LIN {X 0,Y 231.283,Z 816.098,A -85,B 0,C 180,E1 32036.153,E2 32036.153} C_VEL
LIN {X 0,Y 232.3,Z 814.541,A -85,B 0,C 180,E1 32036.256,E2 32036.256} C_VEL
LIN {X 0,Y 232.997,Z 811.859,A -85,B 0,C 180,E1 32038.132,E2 32038.132} C_VEL
LIN {X 0,Y 233.164,Z 810.301,A -85,B 0,C 180,E1 32039.995,E2 32039.995} C_VEL
LIN {X 0,Y 231.964,Z 810.617,A -85,B 0,C 180,E1 32043.74,E2 32043.74} C_VEL
LIN {X 0,Y 228.908,Z 815.493,A -85,B 0,C 180,E1 32049.516,E2 32049.516} C_VEL
LIN {X 0,Y 226.036,Z 820.81,A -85,B 0,C 180,E1 32052.805,E2 32052.805} C_VEL
LIN {X 0,Y 201.465,Z 849.972,A -85,B 0,C 180,E1 32056.439,E2 32056.439} C_VEL
LIN {X 0,Y 175.055,Z 874.28,A -85,B 0,C 180,E1 32061.454,E2 32061.454} C_VEL
LIN {X 0,Y 147.098,Z 894.32,A -85,B 0,C 180,E1 32068.856,E2 32068.856} C_VEL
LIN {X 0,Y 119.761,Z 909.714,A -85,B 0,C 180,E1 32080.583,E2 32080.583} C_VEL
LIN {X 0,Y 99.708,Z 918.948,A -85,B 0,C 180,E1 32096.749,E2 32096.749} C_VEL
LIN {X 0,Y 88.361,Z 923.461,A -85,B 0,C 180,E1 32120.099,E2 32120.099} C_VEL
LIN {X 0,Y 88.441,Z 923.431,A -85,B 0,C 180,E1 32139.837,E2 32139.837} C_VEL
LIN {X 0,Y 99.926,Z 918.782,A -85,B 0,C 180,E1 32163.44,E2 32163.44} C_VEL
LIN {X 0,Y 119.785,Z 909.607,A -85,B 0,C 180,E1 32179.342,E2 32179.342} C_VEL
LIN {X 0,Y 119.619,Z 909.301,A -85,B 0,C 180,E1 32180.724,E2 32180.724} C_VEL
LIN {X 0,Y 90.219,Z 920.421,A -85,B 0,C 180,E1 32221.835,E2 32221.835} C_VEL
LIN {X 0,Y 87.807,Z 924.074,A -85,B 0,C 180,E1 32232.793,E2 32232.793} C_VEL
LIN {X 0,Y 88.883,Z 927.566,A -85,B 0,C 180,E1 32243.903,E2 32243.903} C_VEL
LIN {X 0,Y 99.549,Z 930.781,A -85,B 0,C 180,E1 32256.148,E2 32256.148} C_VEL
LIN {X 0,Y 97.42,Z 932.429,A -85,B 0,C 180,E1 32258.992,E2 32258.992} C_VEL
LIN {X 0,Y 80.593,Z 941.329,A -85,B 0,C 180,E1 32281.998,E2 32281.998} C_VEL
LIN {X 0,Y 77.652,Z 944.052,A -85,B 0,C 180,E1 32298.779,E2 32298.779} C_VEL
LIN {X 0,Y 78.572,Z 944.794,A -85,B 0,C 180,E1 32310.03,E2 32310.03} C_VEL
LIN {X 0,Y 78.579,Z 942.435,A -85,B 0,C 180,E1 32332.717,E2 32332.717} C_VEL
LIN {X 0,Y 92.775,Z 933.853,A -85,B 0,C 180,E1 32359.206,E2 32359.206} C_VEL
LIN {X 0,Y 118.649,Z 919.574,A -85,B 0,C 180,E1 32376.148,E2 32376.148} C_VEL
LIN {X 0,Y 147.805,Z 900.768,A -85,B 0,C 180,E1 32385.844,E2 32385.844} C_VEL
LIN {X 0,Y 177.973,Z 876.597,A -85,B 0,C 180,E1 32391.869,E2 32391.869} C_VEL
LIN {X 0,Y 206.02,Z 847.904,A -85,B 0,C 180,E1 32395.688,E2 32395.688} C_VEL
LIN {X 0,Y 227.481,Z 820.1,A -85,B 0,C 180,E1 32397.863,E2 32397.863} C_VEL
LIN {X 0,Y 228.556,Z 817.821,A -85,B 0,C 180,E1 32398.934,E2 32398.934} C_VEL
LIN {X 0,Y 228.688,Z 816.963,A -85,B 0,C 180,E1 32399.995,E2 32399.995} C_VEL
LIN {X 0,Y 227.313,Z 817.302,A -85,B 0,C 180,E1 32403.816,E2 32403.816} C_VEL
LIN {X 0,Y 223.822,Z 822.315,A -85,B 0,C 180,E1 32409.605,E2 32409.605} C_VEL
LIN {X 0,Y 221.659,Z 825.693,A -85,B 0,C 180,E1 32411.2,E2 32411.2} C_VEL
LIN {X 0,Y 195.972,Z 854.587,A -85,B 0,C 180,E1 32414.832,E2 32414.832} C_VEL
LIN {X 0,Y 167.376,Z 879.131,A -85,B 0,C 180,E1 32420.037,E2 32420.037} C_VEL
LIN {X 0,Y 140.432,Z 897.198,A -85,B 0,C 180,E1 32427.072,E2 32427.072} C_VEL
LIN {X 0,Y 112.214,Z 911.987,A -85,B 0,C 180,E1 32439.033,E2 32439.033} C_VEL
LIN {X 0,Y 92.464,Z 920.215,A -85,B 0,C 180,E1 32454.982,E2 32454.982} C_VEL
LIN {X 0,Y 80.648,Z 924.449,A -85,B 0,C 180,E1 32479.141,E2 32479.141} C_VEL
LIN {X 0,Y 80.725,Z 924.423,A -85,B 0,C 180,E1 32500.788,E2 32500.788} C_VEL
LIN {X 0,Y 92.642,Z 920.094,A -85,B 0,C 180,E1 32525.175,E2 32525.175} C_VEL
LIN {X 0,Y 109.719,Z 912.985,A -85,B 0,C 180,E1 32539.39,E2 32539.39} C_VEL
LIN {X 0,Y 108.72,Z 912.974,A -85,B 0,C 180,E1 32541.182,E2 32541.182} C_VEL
LIN {X 0,Y 88.883,Z 927.566,A -85,B 0,C 180,E1 32603.903,E2 32603.903} C_VEL
LIN {X 0,Y 91.046,Z 929.778,A -85,B 0,C 180,E1 32610.655,E2 32610.655} C_VEL
LIN {X 0,Y 89.329,Z 932.69,A -85,B 0,C 180,E1 32617.152,E2 32617.152} C_VEL
LIN {X 0,Y 87.849,Z 933.503,A -85,B 0,C 180,E1 32618.803,E2 32618.803} C_VEL
LIN {X 0,Y 71.627,Z 941.461,A -85,B 0,C 180,E1 32645.008,E2 32645.008} C_VEL
LIN {X 0,Y 70.618,Z 943.791,A -85,B 0,C 180,E1 32670.034,E2 32670.034} C_VEL
LIN {X 0,Y 71.144,Z 941.405,A -85,B 0,C 180,E1 32695.248,E2 32695.248} C_VEL
LIN {X 0,Y 87.583,Z 932.779,A -85,B 0,C 180,E1 32723.316,E2 32723.316} C_VEL
LIN {X 0,Y 115.54,Z 918.483,A -85,B 0,C 180,E1 32739.919,E2 32739.919} C_VEL
LIN {X 0,Y 146.614,Z 899.19,A -85,B 0,C 180,E1 32749.136,E2 32749.136} C_VEL
LIN {X 0,Y 178.554,Z 874.062,A -85,B 0,C 180,E1 32754.74,E2 32754.74} C_VEL
LIN {X 0,Y 206.65,Z 845.496,A -85,B 0,C 180,E1 32758.072,E2 32758.072} C_VEL
LIN {X 0,Y 222.734,Z 825.385,A -85,B 0,C 180,E1 32759.528,E2 32759.528} C_VEL
LIN {X 0,Y 223.946,Z 823.43,A -85,B 0,C 180,E1 32759.995,E2 32759.995} C_VEL
LIN {X 0,Y 222.493,Z 823.879,A -85,B 0,C 180,E1 32763.899,E2 32763.899} C_VEL
LIN {X 0,Y 219.282,Z 827.949,A -85,B 0,C 180,E1 32768.768,E2 32768.768} C_VEL
LIN {X 0,Y 217.386,Z 830.343,A -85,B 0,C 180,E1 32769.537,E2 32769.537} C_VEL
LIN {X 0,Y 190.615,Z 858.942,A -85,B 0,C 180,E1 32773.101,E2 32773.101} C_VEL
LIN {X 0,Y 161.481,Z 882.675,A -85,B 0,C 180,E1 32778.139,E2 32778.139} C_VEL
LIN {X 0,Y 130.785,Z 901.732,A -85,B 0,C 180,E1 32786.079,E2 32786.079} C_VEL
LIN {X 0,Y 102.133,Z 915.175,A -85,B 0,C 180,E1 32798.806,E2 32798.806} C_VEL
LIN {X 0,Y 82.386,Z 922.477,A -85,B 0,C 180,E1 32816.478,E2 32816.478} C_VEL
LIN {X 0,Y 72.949,Z 925.439,A -85,B 0,C 180,E1 32837.979,E2 32837.979} C_VEL
LIN {X 0,Y 73.048,Z 925.413,A -85,B 0,C 180,E1 32861.938,E2 32861.938} C_VEL
LIN {X 0,Y 86.324,Z 921.102,A -85,B 0,C 180,E1 32888.188,E2 32888.188} C_VEL
LIN {X 0,Y 99.662,Z 916.141,A -85,B 0,C 180,E1 32899.442,E2 32899.442} C_VEL
LIN {X 0,Y 97.848,Z 916.351,A -85,B 0,C 180,E1 32901.751,E2 32901.751} C_VEL
LIN {X 0,Y 90.297,Z 932.103,A -85,B 0,C 180,E1 32975.972,E2 32975.972} C_VEL
LIN {X 0,Y 87.849,Z 933.503,A -85,B 0,C 180,E1 32978.803,E2 32978.803} C_VEL
LIN {X 0,Y 75.565,Z 937.247,A -85,B 0,C 180,E1 32987.238,E2 32987.238} C_VEL
LIN {X 0,Y 65.402,Z 939.87,A -85,B 0,C 180,E1 32998.741,E2 32998.741} C_VEL
LIN {X 0,Y 62.681,Z 942.791,A -85,B 0,C 180,E1 33030.038,E2 33030.038} C_VEL
LIN {X 0,Y 63.847,Z 940.368,A -85,B 0,C 180,E1 33058.378,E2 33058.378} C_VEL
LIN {X 0,Y 82.635,Z 931.823,A -85,B 0,C 180,E1 33087.678,E2 33087.678} C_VEL
LIN {X 0,Y 113.083,Z 917.306,A -85,B 0,C 180,E1 33103.951,E2 33103.951} C_VEL
LIN {X 0,Y 145.282,Z 898.069,A -85,B 0,C 180,E1 33112.343,E2 33112.343} C_VEL
LIN {X 0,Y 177.269,Z 873.513,A -85,B 0,C 180,E1 33117.31,E2 33117.31} C_VEL
LIN {X 0,Y 205.431,Z 845.518,A -85,B 0,C 180,E1 33120.246,E2 33120.246} C_VEL
LIN {X 0,Y 217.358,Z 831.322,A -85,B 0,C 180,E1 33121.22,E2 33121.22} C_VEL
LIN {X 0,Y 218.373,Z 829.868,A -85,B 0,C 180,E1 33121.575,E2 33121.575} C_VEL
LIN {X 0,Y 216.429,Z 831.287,A -85,B 0,C 180,E1 33125.53,E2 33125.53} C_VEL
LIN {X 0,Y 214.109,Z 834.024,A -85,B 0,C 180,E1 33127.716,E2 33127.716} C_VEL
LIN {X 0,Y 187.221,Z 861.636,A -85,B 0,C 180,E1 33131.034,E2 33131.034} C_VEL
LIN {X 0,Y 157.493,Z 884.892,A -85,B 0,C 180,E1 33135.774,E2 33135.774} C_VEL
LIN {X 0,Y 127.517,Z 902.769,A -85,B 0,C 180,E1 33142.896,E2 33142.896} C_VEL
LIN {X 0,Y 97.385,Z 916.188,A -85,B 0,C 180,E1 33155.187,E2 33155.187} C_VEL
LIN {X 0,Y 75.96,Z 923.473,A -85,B 0,C 180,E1 33173.204,E2 33173.204} C_VEL
LIN {X 0,Y 65.299,Z 926.428,A -85,B 0,C 180,E1 33196.545,E2 33196.545} C_VEL
LIN {X 0,Y 65.393,Z 926.404,A -85,B 0,C 180,E1 33223.36,E2 33223.36} C_VEL
LIN {X 0,Y 80.077,Z 922.171,A -85,B 0,C 180,E1 33251.426,E2 33251.426} C_VEL
LIN {X 0,Y 88.712,Z 919.304,A -85,B 0,C 180,E1 33258.986,E2 33258.986} C_VEL
LIN {X 0,Y 89.578,Z 918.903,A -85,B 0,C 180,E1 33260.494,E2 33260.494} C_VEL
LIN {X 0,Y 80.603,Z 933.165,A -85,B 0,C 180,E1 33335.59,E2 33335.59} C_VEL
LIN {X 0,Y 65.402,Z 939.87,A -85,B 0,C 180,E1 33358.741,E2 33358.741} C_VEL
LIN {X 0,Y 59.44,Z 941.678,A -85,B 0,C 180,E1 33373.874,E2 33373.874} C_VEL
LIN {X 0,Y 54.539,Z 941.732,A -85,B 0,C 180,E1 33391.166,E2 33391.166} C_VEL
LIN {X 0,Y 56.81,Z 939.335,A -85,B 0,C 180,E1 33422.287,E2 33422.287} C_VEL
LIN {X 0,Y 79.233,Z 930.482,A -85,B 0,C 180,E1 33453.317,E2 33453.317} C_VEL
LIN {X 0,Y 111.051,Z 916.181,A -85,B 0,C 180,E1 33468.128,E2 33468.128} C_VEL
LIN {X 0,Y 144.414,Z 896.958,A -85,B 0,C 180,E1 33475.586,E2 33475.586} C_VEL
LIN {X 0,Y 177.293,Z 872.162,A -85,B 0,C 180,E1 33479.994,E2 33479.994} C_VEL
LIN {X 0,Y 205.686,Z 844.302,A -85,B 0,C 180,E1 33482.535,E2 33482.535} C_VEL
LIN {X 0,Y 212.464,Z 836.508,A -85,B 0,C 180,E1 33483.015,E2 33483.015} C_VEL
LIN {X 0,Y 211.021,Z 837.726,A -85,B 0,C 180,E1 33485.672,E2 33485.672} C_VEL
LIN {X 0,Y 182.814,Z 865.442,A -85,B 0,C 180,E1 33489.037,E2 33489.037} C_VEL
LIN {X 0,Y 152.029,Z 888.247,A -85,B 0,C 180,E1 33493.587,E2 33493.587} C_VEL
LIN {X 0,Y 121.352,Z 905.407,A -85,B 0,C 180,E1 33500.48,E2 33500.48} C_VEL
LIN {X 0,Y 90.203,Z 918.281,A -85,B 0,C 180,E1 33512.823,E2 33512.823} C_VEL
LIN {X 0,Y 69.819,Z 924.471,A -85,B 0,C 180,E1 33529.334,E2 33529.334} C_VEL
LIN {X 0,Y 57.689,Z 927.418,A -85,B 0,C 180,E1 33554.73,E2 33554.73} C_VEL
LIN {X 0,Y 57.778,Z 927.395,A -85,B 0,C 180,E1 33585.161,E2 33585.161} C_VEL
LIN {X 0,Y 74.368,Z 923.176,A -85,B 0,C 180,E1 33615.442,E2 33615.442} C_VEL
LIN {X 0,Y 79.297,Z 921.703,A -85,B 0,C 180,E1 33619.799,E2 33619.799} C_VEL
LIN {X 0,Y 61.032,Z 930.524,A -85,B 0,C 180,E1 33674.39,E2 33674.39} C_VEL
LIN {X 0,Y 70.568,Z 933.916,A -85,B 0,C 180,E1 33694.568,E2 33694.568} C_VEL
LIN {X 0,Y 68.147,Z 935.33,A -85,B 0,C 180,E1 33698.959,E2 33698.959} C_VEL
LIN {X 0,Y 54.26,Z 941.014,A -85,B 0,C 180,E1 33733.831,E2 33733.831} C_VEL
LIN {X 0,Y 54.539,Z 941.732,A -85,B 0,C 180,E1 33751.166,E2 33751.166} C_VEL
LIN {X 0,Y 51.278,Z 940.81,A -85,B 0,C 180,E1 33764.904,E2 33764.904} C_VEL
LIN {X 0,Y 50.905,Z 937.953,A -85,B 0,C 180,E1 33789.635,E2 33789.635} C_VEL
LIN {X 0,Y 76.86,Z 929.056,A -85,B 0,C 180,E1 33819.536,E2 33819.536} C_VEL
LIN {X 0,Y 110.439,Z 914.69,A -85,B 0,C 180,E1 33832.57,E2 33832.57} C_VEL
LIN {X 0,Y 145.896,Z 894.56,A -85,B 0,C 180,E1 33839.158,E2 33839.158} C_VEL
LIN {X 0,Y 179.314,Z 869.458,A -85,B 0,C 180,E1 33842.814,E2 33842.814} C_VEL
LIN {X 0,Y 198.983,Z 850.837,A -85,B 0,C 180,E1 33844.361,E2 33844.361} C_VEL
LIN {X 0,Y 197.748,Z 851.989,A -85,B 0,C 180,E1 33844.923,E2 33844.923} C_VEL
LIN {X 0,Y 168.427,Z 876.998,A -85,B 0,C 180,E1 33848.178,E2 33848.178} C_VEL
LIN {X 0,Y 136.883,Z 897.299,A -85,B 0,C 180,E1 33852.968,E2 33852.968} C_VEL
LIN {X 0,Y 103.751,Z 912.967,A -85,B 0,C 180,E1 33861.219,E2 33861.219} C_VEL
LIN {X 0,Y 74.486,Z 922.762,A -85,B 0,C 180,E1 33875.487,E2 33875.487} C_VEL
LIN {X 0,Y 55.629,Z 927.34,A -85,B 0,C 180,E1 33896.941,E2 33896.941} C_VEL
LIN {X 0,Y 48.588,Z 928.763,A -85,B 0,C 180,E1 33929.951,E2 33929.951} C_VEL
LIN {X 0,Y 62.689,Z 925.769,A -85,B 0,C 180,E1 33973.56,E2 33973.56} C_VEL
LIN {X 0,Y 68.76,Z 924.236,A -85,B 0,C 180,E1 33980.9,E2 33980.9} C_VEL
LIN {X 0,Y 60.712,Z 934.548,A -85,B 0,C 180,E1 34053.502,E2 34053.502} C_VEL
LIN {X 0,Y 58.394,Z 935.838,A -85,B 0,C 180,E1 34058.947,E2 34058.947} C_VEL
LIN {X 0,Y 46.086,Z 940.484,A -85,B 0,C 180,E1 34100.589,E2 34100.589} C_VEL
LIN {X 0,Y 46.77,Z 940.785,A -85,B 0,C 180,E1 34110.051,E2 34110.051} C_VEL
LIN {X 0,Y 50.905,Z 937.953,A -85,B 0,C 180,E1 34149.635,E2 34149.635} C_VEL
LIN {X 0,Y 56.414,Z 934.774,A -85,B 0,C 180,E1 34167.148,E2 34167.148} C_VEL
LIN {X 0,Y 65.816,Z 930.795,A -85,B 0,C 180,E1 34180.645,E2 34180.645} C_VEL
LIN {X 0,Y 98.93,Z 918.458,A -85,B 0,C 180,E1 34194.35,E2 34194.35} C_VEL
LIN {X 0,Y 136.444,Z 899.357,A -85,B 0,C 180,E1 34201.28,E2 34201.28} C_VEL
LIN {X 0,Y 169.433,Z 876.806,A -85,B 0,C 180,E1 34204.675,E2 34204.675} C_VEL
LIN {X 0,Y 171.885,Z 874.872,A -85,B 0,C 180,E1 34205.05,E2 34205.05} C_VEL
LIN {X 0,Y 138.216,Z 896.785,A -85,B 0,C 180,E1 34209.271,E2 34209.271} C_VEL
LIN {X 0,Y 102.127,Z 913.607,A -85,B 0,C 180,E1 34216.792,E2 34216.792} C_VEL
LIN {X 0,Y 70.215,Z 923.773,A -85,B 0,C 180,E1 34230.258,E2 34230.258} C_VEL
LIN {X 0,Y 49.243,Z 928.334,A -85,B 0,C 180,E1 34251.958,E2 34251.958} C_VEL
LIN {X 0,Y 40.742,Z 929.753,A -85,B 0,C 180,E1 34289.941,E2 34289.941} C_VEL
LIN {X 0,Y 49.255,Z 928.304,A -85,B 0,C 180,E1 34327.909,E2 34327.909} C_VEL
LIN {X 0,Y 58.774,Z 926.416,A -85,B 0,C 180,E1 34340.596,E2 34340.596} C_VEL
LIN {X 0,Y 50.601,Z 934.935,A -85,B 0,C 180,E1 34411.62,E2 34411.62} C_VEL
LIN {X 0,Y 50.997,Z 935.557,A -85,B 0,C 180,E1 34415.455,E2 34415.455} C_VEL
LIN {X 0,Y 39.067,Z 938.982,A -85,B 0,C 180,E1 34447.246,E2 34447.246} C_VEL
LIN {X 0,Y 38.792,Z 939.779,A -85,B 0,C 180,E1 34470.062,E2 34470.062} C_VEL
LIN {X 0,Y 46.182,Z 936.566,A -85,B 0,C 180,E1 34518.97,E2 34518.97} C_VEL
LIN {X 0,Y 65.816,Z 930.795,A -85,B 0,C 180,E1 34540.645,E2 34540.645} C_VEL
LIN {X 0,Y 77.565,Z 926.098,A -85,B 0,C 180,E1 34550.398,E2 34550.398} C_VEL
LIN {X 0,Y 90.669,Z 920.51,A -85,B 0,C 180,E1 34557.428,E2 34557.428} C_VEL
LIN {X 0,Y 127.54,Z 903.494,A -85,B 0,C 180,E1 34563.742,E2 34563.742} C_VEL
LIN {X 0,Y 141.711,Z 895.332,A -85,B 0,C 180,E1 34565.203,E2 34565.203} C_VEL
LIN {X 0,Y 108.01,Z 911.611,A -85,B 0,C 180,E1 34570.775,E2 34570.775} C_VEL
LIN {X 0,Y 73.164,Z 923.143,A -85,B 0,C 180,E1 34581.172,E2 34581.172} C_VEL
LIN {X 0,Y 43.324,Z 929.331,A -85,B 0,C 180,E1 34605.538,E2 34605.538} C_VEL
LIN {X 0,Y 32.912,Z 930.74,A -85,B 0,C 180,E1 34649.927,E2 34649.927} C_VEL
LIN {X 0,Y 48.15,Z 928.49,A -85,B 0,C 180,E1 34701.036,E2 34701.036} C_VEL
LIN {X 0,Y 41.57,Z 935.37,A -85,B 0,C 180,E1 34771.57,E2 34771.57} C_VEL
LIN {X 0,Y 38.891,Z 936.328,A -85,B 0,C 180,E1 34778.91,E2 34778.91} C_VEL
LIN {X 0,Y 30.804,Z 938.772,A -85,B 0,C 180,E1 34830.078,E2 34830.078} C_VEL
LIN {X 0,Y 41.246,Z 935.517,A -85,B 0,C 180,E1 34887.633,E2 34887.633} C_VEL
LIN {X 0,Y 76.334,Z 925.73,A -85,B 0,C 180,E1 34913.231,E2 34913.231} C_VEL
LIN {X 0,Y 90.669,Z 920.51,A -85,B 0,C 180,E1 34917.428,E2 34917.428} C_VEL
LIN {X 0,Y 99.273,Z 916.582,A -85,B 0,C 180,E1 34921.763,E2 34921.763} C_VEL
LIN {X 0,Y 108.215,Z 912.239,A -85,B 0,C 180,E1 34925.308,E2 34925.308} C_VEL
LIN {X 0,Y 110.92,Z 910.99,A -85,B 0,C 180,E1 34925.644,E2 34925.644} C_VEL
LIN {X 0,Y 77.766,Z 922.338,A -85,B 0,C 180,E1 34932.906,E2 34932.906} C_VEL
LIN {X 0,Y 50.325,Z 928.47,A -85,B 0,C 180,E1 34945.3,E2 34945.3} C_VEL
LIN {X 0,Y 28.637,Z 931.382,A -85,B 0,C 180,E1 34977.957,E2 34977.957} C_VEL
LIN {X 0,Y 25.065,Z 931.729,A -85,B 0,C 180,E1 35009.905,E2 35009.905} C_VEL
LIN {X 0,Y 35.062,Z 930.658,A -85,B 0,C 180,E1 35057.892,E2 35057.892} C_VEL
LIN {X 0,Y 36.419,Z 930.586,A -85,B 0,C 180,E1 35063.849,E2 35063.849} C_VEL
LIN {X 0,Y 31.73,Z 935.383,A -85,B 0,C 180,E1 35128.557,E2 35128.557} C_VEL
LIN {X 0,Y 25.014,Z 936.951,A -85,B 0,C 180,E1 35152.838,E2 35152.838} C_VEL
LIN {X 0,Y 22.799,Z 937.763,A -85,B 0,C 180,E1 35190.105,E2 35190.105} C_VEL
LIN {X 0,Y 34.079,Z 935.154,A -85,B 0,C 180,E1 35253.572,E2 35253.572} C_VEL
LIN {X 0,Y 68.303,Z 926.94,A -85,B 0,C 180,E1 35277.278,E2 35277.278} C_VEL
LIN {X 0,Y 108.215,Z 912.239,A -85,B 0,C 180,E1 35285.308,E2 35285.308} C_VEL
LIN {X 0,Y 101.377,Z 914.887,A -85,B 0,C 180,E1 35286.476,E2 35286.476} C_VEL
LIN {X 0,Y 69.327,Z 925.196,A -85,B 0,C 180,E1 35288.959,E2 35288.959} C_VEL
LIN {X 0,Y 65.375,Z 926.062,A -85,B 0,C 180,E1 35289.9,E2 35289.9} C_VEL
LIN {X 0,Y 33.941,Z 931.318,A -85,B 0,C 180,E1 35306.609,E2 35306.609} C_VEL
LIN {X 0,Y 17.235,Z 932.716,A -85,B 0,C 180,E1 35369.861,E2 35369.861} C_VEL
LIN {X 0,Y 22.411,Z 932.345,A -85,B 0,C 180,E1 35412.395,E2 35412.395} C_VEL
LIN {X 0,Y 26.196,Z 932.155,A -85,B 0,C 180,E1 35424.721,E2 35424.721} C_VEL
LIN {X 0,Y 22.085,Z 935.233,A -85,B 0,C 180,E1 35483.114,E2 35483.114} C_VEL
LIN {X 0,Y 19.021,Z 935.894,A -85,B 0,C 180,E1 35497.402,E2 35497.402} C_VEL
LIN {X 0,Y 14.756,Z 936.749,A -85,B 0,C 180,E1 35550.162,E2 35550.162} C_VEL
LIN {X 0,Y 31.14,Z 934.132,A -85,B 0,C 180,E1 35627.035,E2 35627.035} C_VEL
LIN {X 0,Y 68.415,Z 925.875,A -85,B 0,C 180,E1 35644.258,E2 35644.258} C_VEL
LIN {X 0,Y 76.185,Z 923.591,A -85,B 0,C 180,E1 35645.748,E2 35645.748} C_VEL
LIN {X 0,Y 76.392,Z 923.354,A -85,B 0,C 180,E1 35647.125,E2 35647.125} C_VEL
LIN {X 0,Y 65.375,Z 926.062,A -85,B 0,C 180,E1 35649.9,E2 35649.9} C_VEL
LIN {X 0,Y 52.547,Z 928.896,A -85,B 0,C 180,E1 35650.66,E2 35650.66} C_VEL
LIN {X 0,Y 30.988,Z 932.987,A -85,B 0,C 180,E1 35642.658,E2 35642.658} C_VEL
LIN {X 0,Y 6.73,Z 935.737,A -85,B 0,C 180,E1 35550.355,E2 35550.355} C_VEL
LIN {X 0,Y 10.702,Z 935.3,A -85,B 0,C 180,E1 35485.965,E2 35485.965} C_VEL
LIN {X 0,Y 12.942,Z 934.866,A -85,B 0,C 180,E1 35470.472,E2 35470.472} C_VEL
LIN {X 0,Y 15.186,Z 933.592,A -85,B 0,C 180,E1 35430.164,E2 35430.164} C_VEL
LIN {X 0,Y 11.802,Z 933.603,A -85,B 0,C 180,E1 35409.674,E2 35409.674} C_VEL
LIN {X 0,Y 31.222,Z 932.314,A -85,B 0,C 180,E1 35293.607,E2 35293.607} C_VEL
LIN {X 0,Y 43.975,Z 930.842,A -85,B 0,C 180,E1 35287.026,E2 35287.026} C_VEL
LIN {X 0,Y 30.988,Z 932.987,A -85,B 0,C 180,E1 35282.658,E2 35282.658} C_VEL
LIN {X 0,Y 29.357,Z 934.962,A -85,B 0,C 180,E1 35281.831,E2 35281.831} C_VEL
LIN {X 0,Y 29.357,Z 1012.5,A -85,B 0,C 180,E1 35281.831,E2 35281.831} C_VEL
LIN {X 0,Y 29.357,Z 1012.5,A -85,B 0,C 180,E1 35281.831,E2 35281.831}

QRS_NEXT_CUT()
PTP {E1 35457.186,E2 35457.186}
PTP {X 0,Y 759.911,A -85,B 0,C 180,E1 35457.186,E2 35457.186,E3 0,E4 0,E5 0,E6 0}
QRS_SPEED_INIT()
LIN {X 0,Y 759.911,Z 1012.5,A -85,B 0,C 180,E1 35457.186,E2 35457.186,E3 0,E4 0,E5 0,E6 0} C_VEL
LIN {X 0,Y 759.911,Z 859.359,A -85,B 0,C 180,E1 35457.186,E2 35457.186} C_VEL
LIN {X 0,Y 759.911,Z 850.88,A -85,B 0,C 180,E1 35457.186,E2 35457.186} C_VEL
LIN {X 0,Y 759.915,Z 848.921,A -85,B 0,C 180,E1 35457.065,E2 35457.065} C_VEL
LIN {X 0,Y 759.916,Z 844.691,A -85,B 0,C 180,E1 35455.699,E2 35455.699} C_VEL
LIN {X 0,Y 759.912,Z 838.727,A -85,B 0,C 180,E1 35454.337,E2 35454.337} C_VEL
LIN {X 0,Y 759.916,Z 830.826,A -85,B 0,C 180,E1 35452.971,E2 35452.971} C_VEL
LIN {X 0,Y 759.916,Z 821.375,A -85,B 0,C 180,E1 35451.678,E2 35451.678} C_VEL
LIN {X 0,Y 759.915,Z 810.407,A -85,B 0,C 180,E1 35450.457,E2 35450.457} C_VEL
LIN {X 0,Y 759.914,Z 797.91,A -85,B 0,C 180,E1 35449.308,E2 35449.308} C_VEL
LIN {X 0,Y 759.916,Z 783.678,A -85,B 0,C 180,E1 35448.223,E2 35448.223} C_VEL
LIN {X 0,Y 759.918,Z 768.565,A -85,B 0,C 180,E1 35447.268,E2 35447.268} C_VEL
LIN {X 0,Y 759.918,Z 753.017,A -85,B 0,C 180,E1 35446.455,E2 35446.455} C_VEL
LIN {X 0,Y 759.892,Z 736.694,A -85,B 0,C 180,E1 35445.755,E2 35445.755} C_VEL
LIN {X 0,Y 759.918,Z 719.642,A -85,B 0,C 180,E1 35445.172,E2 35445.172} C_VEL
LIN {X 0,Y 759.913,Z 702.22,A -85,B 0,C 180,E1 35444.713,E2 35444.713} C_VEL
LIN {X 0,Y 759.911,Z 683.596,A -85,B 0,C 180,E1 35444.364,E2 35444.364} C_VEL
LIN {X 0,Y 759.901,Z 658.001,A -85,B 0,C 180,E1 35444.077,E2 35444.077} C_VEL
LIN {X 0,Y 759.864,Z 469.775,A -85,B 0,C 180,E1 35442.244,E2 35442.244} C_VEL
LIN {X 0,Y 759.9,Z 416.635,A -85,B 0,C 180,E1 35439.593,E2 35439.593} C_VEL
LIN {X 0,Y 759.918,Z 361.495,A -85,B 0,C 180,E1 35436.791,E2 35436.791} C_VEL
LIN {X 0,Y 759.91,Z 307.45,A -85,B 0,C 180,E1 35433.987,E2 35433.987} C_VEL
LIN {X 0,Y 759.913,Z 254.157,A -85,B 0,C 180,E1 35431.163,E2 35431.163} C_VEL
LIN {X 0,Y 759.884,Z 202.297,A -85,B 0,C 180,E1 35428.359,E2 35428.359} C_VEL
LIN {X 0,Y 759.874,Z 190.577,A -85,B 0,C 180,E1 35427.707,E2 35427.707} C_VEL
LIN {X 0,Y 759.897,Z 190.571,A -85,B 0,C 180,E1 35424.899,E2 35424.899} C_VEL
LIN {X 0,Y 759.895,Z 190.577,A -85,B 0,C 180,E1 35421.989,E2 35421.989} C_VEL
LIN {X 0,Y 759.84,Z 190.578,A -85,B 0,C 180,E1 35419.354,E2 35419.354} C_VEL
LIN {X 0,Y 759.917,Z 190.569,A -85,B 0,C 180,E1 35416.515,E2 35416.515} C_VEL
LIN {X 0,Y 759.911,Z 190.578,A -85,B 0,C 180,E1 35413.589,E2 35413.589} C_VEL
LIN {X 0,Y 759.882,Z 190.572,A -85,B 0,C 180,E1 35410.743,E2 35410.743} C_VEL
LIN {X 0,Y 759.843,Z 190.578,A -85,B 0,C 180,E1 35407.823,E2 35407.823} C_VEL
LIN {X 0,Y 759.881,Z 190.577,A -85,B 0,C 180,E1 35405.286,E2 35405.286} C_VEL
LIN {X 0,Y 759.897,Z 190.758,A -85,B 0,C 180,E1 35402.716,E2 35402.716} C_VEL
LIN {X 0,Y 759.899,Z 231.312,A -85,B 0,C 180,E1 35400.001,E2 35400.001} C_VEL
LIN {X 0,Y 759.904,Z 273.516,A -85,B 0,C 180,E1 35397.252,E2 35397.252} C_VEL
LIN {X 0,Y 759.912,Z 304.464,A -85,B 0,C 180,E1 35395.291,E2 35395.291} C_VEL
LIN {X 0,Y 759.918,Z 592.91,A -85,B 0,C 180,E1 35392.37,E2 35392.37} C_VEL
LIN {X 0,Y 759.914,Z 615.626,A -85,B 0,C 180,E1 35392.085,E2 35392.085} C_VEL
LIN {X 0,Y 759.913,Z 637.423,A -85,B 0,C 180,E1 35391.679,E2 35391.679} C_VEL
LIN {X 0,Y 759.909,Z 657.419,A -85,B 0,C 180,E1 35391.173,E2 35391.173} C_VEL
LIN {X 0,Y 759.905,Z 678.887,A -85,B 0,C 180,E1 35390.488,E2 35390.488} C_VEL
LIN {X 0,Y 759.918,Z 698.468,A -85,B 0,C 180,E1 35389.725,E2 35389.725} C_VEL
LIN {X 0,Y 759.917,Z 717.218,A -85,B 0,C 180,E1 35388.846,E2 35388.846} C_VEL
LIN {X 0,Y 759.915,Z 736.006,A -85,B 0,C 180,E1 35387.814,E2 35387.814} C_VEL
LIN {X 0,Y 759.911,Z 753.642,A -85,B 0,C 180,E1 35386.683,E2 35386.683} C_VEL
LIN {X 0,Y 759.912,Z 770.137,A -85,B 0,C 180,E1 35385.453,E2 35385.453} C_VEL
LIN {X 0,Y 759.919,Z 785.295,A -85,B 0,C 180,E1 35384.131,E2 35384.131} C_VEL
LIN {X 0,Y 759.913,Z 798.741,A -85,B 0,C 180,E1 35382.771,E2 35382.771} C_VEL
LIN {X 0,Y 759.912,Z 811.161,A -85,B 0,C 180,E1 35381.306,E2 35381.306} C_VEL
LIN {X 0,Y 759.912,Z 821.569,A -85,B 0,C 180,E1 35379.849,E2 35379.849} C_VEL
LIN {X 0,Y 759.907,Z 830.684,A -85,B 0,C 180,E1 35378.314,E2 35378.314} C_VEL
LIN {X 0,Y 759.898,Z 838.372,A -85,B 0,C 180,E1 35376.725,E2 35376.725} C_VEL
LIN {X 0,Y 759.904,Z 844.26,A -85,B 0,C 180,E1 35375.133,E2 35375.133} C_VEL
LIN {X 0,Y 759.914,Z 848.686,A -85,B 0,C 180,E1 35373.47,E2 35373.47} C_VEL
LIN {X 0,Y 759.918,Z 851.442,A -85,B 0,C 180,E1 35371.81,E2 35371.81} C_VEL
LIN {X 0,Y 759.908,Z 852.45,A -85,B 0,C 180,E1 35370.151,E2 35370.151} C_VEL
LIN {X 0,Y 759.899,Z 851.787,A -85,B 0,C 180,E1 35368.492,E2 35368.492} C_VEL
LIN {X 0,Y 759.896,Z 849.505,A -85,B 0,C 180,E1 35366.832,E2 35366.832} C_VEL
LIN {X 0,Y 759.902,Z 845.701,A -85,B 0,C 180,E1 35365.245,E2 35365.245} C_VEL
LIN {X 0,Y 759.913,Z 840.243,A -85,B 0,C 180,E1 35363.654,E2 35363.654} C_VEL
LIN {X 0,Y 759.911,Z 833.15,A -85,B 0,C 180,E1 35362.059,E2 35362.059} C_VEL
LIN {X 0,Y 759.903,Z 824.561,A -85,B 0,C 180,E1 35360.533,E2 35360.533} C_VEL
LIN {X 0,Y 759.903,Z 814.081,A -85,B 0,C 180,E1 35358.992,E2 35358.992} C_VEL
LIN {X 0,Y 759.908,Z 802.385,A -85,B 0,C 180,E1 35357.538,E2 35357.538} C_VEL
LIN {X 0,Y 759.906,Z 789.125,A -85,B 0,C 180,E1 35356.144,E2 35356.144} C_VEL
LIN {X 0,Y 759.911,Z 774.48,A -85,B 0,C 180,E1 35354.821,E2 35354.821} C_VEL
LIN {X 0,Y 759.916,Z 757.861,A -85,B 0,C 180,E1 35353.528,E2 35353.528} C_VEL
LIN {X 0,Y 759.917,Z 740.817,A -85,B 0,C 180,E1 35352.384,E2 35352.384} C_VEL
LIN {X 0,Y 759.915,Z 722.406,A -85,B 0,C 180,E1 35351.33,E2 35351.33} C_VEL
LIN {X 0,Y 759.917,Z 703.45,A -85,B 0,C 180,E1 35350.409,E2 35350.409} C_VEL
LIN {X 0,Y 759.916,Z 683.635,A -85,B 0,C 180,E1 35349.593,E2 35349.593} C_VEL
LIN {X 0,Y 759.917,Z 662.813,A -85,B 0,C 180,E1 35348.891,E2 35348.891} C_VEL
LIN {X 0,Y 759.907,Z 642.122,A -85,B 0,C 180,E1 35348.341,E2 35348.341} C_VEL
LIN {X 0,Y 759.915,Z 621.37,A -85,B 0,C 180,E1 35347.915,E2 35347.915} C_VEL
LIN {X 0,Y 759.917,Z 600.246,A -85,B 0,C 180,E1 35347.619,E2 35347.619} C_VEL
LIN {X 0,Y 759.913,Z 307.626,A -85,B 0,C 180,E1 35344.651,E2 35344.651} C_VEL
LIN {X 0,Y 759.917,Z 303.957,A -85,B 0,C 180,E1 35344.599,E2 35344.599} C_VEL
LIN {X 0,Y 759.919,Z 257.758,A -85,B 0,C 180,E1 35341.641,E2 35341.641} C_VEL
LIN {X 0,Y 759.889,Z 216.102,A -85,B 0,C 180,E1 35338.9,E2 35338.9} C_VEL
LIN {X 0,Y 759.875,Z 190.573,A -85,B 0,C 180,E1 35337.171,E2 35337.171} C_VEL
LIN {X 0,Y 759.906,Z 190.578,A -85,B 0,C 180,E1 35334.407,E2 35334.407} C_VEL
LIN {X 0,Y 759.899,Z 190.566,A -85,B 0,C 180,E1 35331.407,E2 35331.407} C_VEL
LIN {X 0,Y 759.893,Z 190.575,A -85,B 0,C 180,E1 35328.558,E2 35328.558} C_VEL
LIN {X 0,Y 759.914,Z 190.565,A -85,B 0,C 180,E1 35325.573,E2 35325.573} C_VEL
LIN {X 0,Y 759.881,Z 190.572,A -85,B 0,C 180,E1 35322.757,E2 35322.757} C_VEL
LIN {X 0,Y 759.901,Z 190.573,A -85,B 0,C 180,E1 35320.021,E2 35320.021} C_VEL
LIN {X 0,Y 759.891,Z 190.567,A -85,B 0,C 180,E1 35317.118,E2 35317.118} C_VEL
LIN {X 0,Y 759.914,Z 190.578,A -85,B 0,C 180,E1 35314.275,E2 35314.275} C_VEL
LIN {X 0,Y 759.912,Z 190.564,A -85,B 0,C 180,E1 35311.315,E2 35311.315} C_VEL
LIN {X 0,Y 759.918,Z 190.577,A -85,B 0,C 180,E1 35308.274,E2 35308.274} C_VEL
LIN {X 0,Y 759.912,Z 190.564,A -85,B 0,C 180,E1 35305.234,E2 35305.234} C_VEL
LIN {X 0,Y 759.91,Z 190.577,A -85,B 0,C 180,E1 35302.269,E2 35302.269} C_VEL
LIN {X 0,Y 759.912,Z 190.564,A -85,B 0,C 180,E1 35299.285,E2 35299.285} C_VEL
LIN {X 0,Y 759.912,Z 190.577,A -85,B 0,C 180,E1 35296.276,E2 35296.276} C_VEL
LIN {X 0,Y 759.901,Z 190.565,A -85,B 0,C 180,E1 35293.313,E2 35293.313} C_VEL
LIN {X 0,Y 759.904,Z 190.574,A -85,B 0,C 180,E1 35290.385,E2 35290.385} C_VEL
LIN {X 0,Y 759.884,Z 190.57,A -85,B 0,C 180,E1 35287.637,E2 35287.637} C_VEL
LIN {X 0,Y 759.903,Z 190.566,A -85,B 0,C 180,E1 35284.831,E2 35284.831} C_VEL
LIN {X 0,Y 759.896,Z 190.575,A -85,B 0,C 180,E1 35281.961,E2 35281.961} C_VEL
LIN {X 0,Y 759.916,Z 190.563,A -85,B 0,C 180,E1 35279.02,E2 35279.02} C_VEL
LIN {X 0,Y 759.9,Z 190.576,A -85,B 0,C 180,E1 35276.001,E2 35276.001} C_VEL
LIN {X 0,Y 759.896,Z 190.565,A -85,B 0,C 180,E1 35273.123,E2 35273.123} C_VEL
LIN {X 0,Y 759.911,Z 190.578,A -85,B 0,C 180,E1 35270.151,E2 35270.151} C_VEL
LIN {X 0,Y 759.874,Z 190.57,A -85,B 0,C 180,E1 35267.383,E2 35267.383} C_VEL
LIN {X 0,Y 759.907,Z 190.569,A -85,B 0,C 180,E1 35264.586,E2 35264.586} C_VEL
LIN {X 0,Y 759.879,Z 190.574,A -85,B 0,C 180,E1 35261.749,E2 35261.749} C_VEL
LIN {X 0,Y 759.887,Z 190.567,A -85,B 0,C 180,E1 35259.028,E2 35259.028} C_VEL
LIN {X 0,Y 759.907,Z 190.577,A -85,B 0,C 180,E1 35256.009,E2 35256.009} C_VEL
LIN {X 0,Y 759.866,Z 190.57,A -85,B 0,C 180,E1 35253.254,E2 35253.254} C_VEL
LIN {X 0,Y 759.912,Z 190.568,A -85,B 0,C 180,E1 35250.521,E2 35250.521} C_VEL
LIN {X 0,Y 759.87,Z 190.574,A -85,B 0,C 180,E1 35247.649,E2 35247.649} C_VEL
LIN {X 0,Y 759.872,Z 190.569,A -85,B 0,C 180,E1 35244.99,E2 35244.99} C_VEL
LIN {X 0,Y 759.918,Z 190.577,A -85,B 0,C 180,E1 35242.086,E2 35242.086} C_VEL
LIN {X 0,Y 759.854,Z 190.573,A -85,B 0,C 180,E1 35239.355,E2 35239.355} C_VEL
LIN {X 0,Y 759.893,Z 190.568,A -85,B 0,C 180,E1 35236.69,E2 35236.69} C_VEL
LIN {X 0,Y 759.873,Z 190.576,A -85,B 0,C 180,E1 35233.696,E2 35233.696} C_VEL
LIN {X 0,Y 759.849,Z 190.572,A -85,B 0,C 180,E1 35231.144,E2 35231.144} C_VEL
LIN {X 0,Y 759.912,Z 190.569,A -85,B 0,C 180,E1 35228.473,E2 35228.473} C_VEL
LIN {X 0,Y 759.86,Z 190.667,A -85,B 0,C 180,E1 35227.583,E2 35227.583} C_VEL
LIN {X 0,Y 759.867,Z 242.061,A -85,B 0,C 180,E1 35225.287,E2 35225.287} C_VEL
LIN {X 0,Y 759.895,Z 298.787,A -85,B 0,C 180,E1 35222.831,E2 35222.831} C_VEL
LIN {X 0,Y 759.917,Z 557.126,A -85,B 0,C 180,E1 35220.027,E2 35220.027} C_VEL
LIN {X 0,Y 759.916,Z 689.995,A -85,B 0,C 180,E1 35218.595,E2 35218.595} C_VEL
LIN {X 0,Y 759.912,Z 714.301,A -85,B 0,C 180,E1 35218.21,E2 35218.21} C_VEL
LIN {X 0,Y 759.907,Z 735.677,A -85,B 0,C 180,E1 35217.742,E2 35217.742} C_VEL
LIN {X 0,Y 759.894,Z 755.109,A -85,B 0,C 180,E1 35217.22,E2 35217.22} C_VEL
LIN {X 0,Y 759.919,Z 777.739,A -85,B 0,C 180,E1 35216.491,E2 35216.491} C_VEL
LIN {X 0,Y 759.916,Z 799.252,A -85,B 0,C 180,E1 35215.651,E2 35215.651} C_VEL
LIN {X 0,Y 759.913,Z 818.66,A -85,B 0,C 180,E1 35214.783,E2 35214.783} C_VEL
LIN {X 0,Y 759.91,Z 841.061,A -85,B 0,C 180,E1 35213.62,E2 35213.62} C_VEL
LIN {X 0,Y 759.911,Z 859.706,A -85,B 0,C 180,E1 35212.513,E2 35212.513} C_VEL
LIN {X 0,Y 759.906,Z 879.524,A -85,B 0,C 180,E1 35211.173,E2 35211.173} C_VEL
LIN {X 0,Y 759.916,Z 896.886,A -85,B 0,C 180,E1 35209.845,E2 35209.845} C_VEL
LIN {X 0,Y 759.907,Z 913.391,A -85,B 0,C 180,E1 35208.409,E2 35208.409} C_VEL
LIN {X 0,Y 759.895,Z 927.948,A -85,B 0,C 180,E1 35206.984,E2 35206.984} C_VEL
LIN {X 0,Y 759.899,Z 942.876,A -85,B 0,C 180,E1 35205.312,E2 35205.312} C_VEL
LIN {X 0,Y 759.91,Z 954.559,A -85,B 0,C 180,E1 35203.816,E2 35203.816} C_VEL
LIN {X 0,Y 759.911,Z 966.786,A -85,B 0,C 180,E1 35201.999,E2 35201.999} C_VEL
LIN {X 0,Y 759.907,Z 975.555,A -85,B 0,C 180,E1 35200.462,E2 35200.462} C_VEL
LIN {X 0,Y 759.883,Z 984.074,A -85,B 0,C 180,E1 35198.704,E2 35198.704} C_VEL
LIN {X 0,Y 759.918,Z 990.726,A -85,B 0,C 180,E1 35196.953,E2 35196.953} C_VEL
LIN {X 0,Y 759.883,Z 995.51,A -85,B 0,C 180,E1 35195.361,E2 35195.361} C_VEL
LIN {X 0,Y 759.919,Z 999.559,A -85,B 0,C 180,E1 35193.47,E2 35193.47} C_VEL
LIN {X 0,Y 759.903,Z 1001.63,A -85,B 0,C 180,E1 35191.81,E2 35191.81} C_VEL
LIN {X 0,Y 759.92,Z 1002.5,A -85,B 0,C 180,E1 35190,E2 35190} C_VEL
LIN {X 0,Y 759.904,Z 1001.63,A -85,B 0,C 180,E1 35188.19,E2 35188.19} C_VEL
LIN {X 0,Y 759.919,Z 999.559,A -85,B 0,C 180,E1 35186.53,E2 35186.53} C_VEL
LIN {X 0,Y 759.883,Z 995.51,A -85,B 0,C 180,E1 35184.639,E2 35184.639} C_VEL
LIN {X 0,Y 759.918,Z 990.725,A -85,B 0,C 180,E1 35183.047,E2 35183.047} C_VEL
LIN {X 0,Y 759.884,Z 983.729,A -85,B 0,C 180,E1 35181.22,E2 35181.22} C_VEL
LIN {X 0,Y 759.907,Z 975.555,A -85,B 0,C 180,E1 35179.538,E2 35179.538} C_VEL
LIN {X 0,Y 759.911,Z 966.785,A -85,B 0,C 180,E1 35178.001,E2 35178.001} C_VEL
LIN {X 0,Y 759.909,Z 954.265,A -85,B 0,C 180,E1 35176.144,E2 35176.144} C_VEL
LIN {X 0,Y 759.9,Z 942.679,A -85,B 0,C 180,E1 35174.664,E2 35174.664} C_VEL
LIN {X 0,Y 759.896,Z 927.17,A -85,B 0,C 180,E1 35172.937,E2 35172.937} C_VEL
LIN {X 0,Y 759.903,Z 912.54,A -85,B 0,C 180,E1 35171.512,E2 35171.512} C_VEL
LIN {X 0,Y 759.917,Z 894.472,A -85,B 0,C 180,E1 35169.964,E2 35169.964} C_VEL
LIN {X 0,Y 759.91,Z 877.578,A -85,B 0,C 180,E1 35168.684,E2 35168.684} C_VEL
LIN {X 0,Y 759.913,Z 857.72,A -85,B 0,C 180,E1 35167.364,E2 35167.364} C_VEL
LIN {X 0,Y 759.91,Z 838.877,A -85,B 0,C 180,E1 35166.257,E2 35166.257} C_VEL
LIN {X 0,Y 759.913,Z 817.007,A -85,B 0,C 180,E1 35165.14,E2 35165.14} C_VEL
LIN {X 0,Y 759.917,Z 798.063,A -85,B 0,C 180,E1 35164.299,E2 35164.299} C_VEL
LIN {X 0,Y 759.912,Z 775.318,A -85,B 0,C 180,E1 35163.425,E2 35163.425} C_VEL
LIN {X 0,Y 759.895,Z 754.005,A -85,B 0,C 180,E1 35162.748,E2 35162.748} C_VEL
LIN {X 0,Y 759.906,Z 734.048,A -85,B 0,C 180,E1 35162.218,E2 35162.218} C_VEL
LIN {X 0,Y 759.917,Z 709.304,A -85,B 0,C 180,E1 35161.7,E2 35161.7} C_VEL
LIN {X 0,Y 759.916,Z 688.273,A -85,B 0,C 180,E1 35161.383,E2 35161.383} C_VEL
LIN {X 0,Y 759.868,Z 431.867,A -85,B 0,C 180,E1 35158.623,E2 35158.623} C_VEL
LIN {X 0,Y 759.895,Z 298.203,A -85,B 0,C 180,E1 35157.151,E2 35157.151} C_VEL
LIN {X 0,Y 759.867,Z 239.96,A -85,B 0,C 180,E1 35154.621,E2 35154.621} C_VEL
LIN {X 0,Y 759.906,Z 190.577,A -85,B 0,C 180,E1 35152.405,E2 35152.405} C_VEL
LIN {X 0,Y 759.909,Z 190.576,A -85,B 0,C 180,E1 35149.512,E2 35149.512} C_VEL
LIN {X 0,Y 759.908,Z 190.578,A -85,B 0,C 180,E1 35146.689,E2 35146.689} C_VEL
LIN {X 0,Y 759.915,Z 190.577,A -85,B 0,C 180,E1 35143.797,E2 35143.797} C_VEL
LIN {X 0,Y 759.909,Z 190.578,A -85,B 0,C 180,E1 35140.94,E2 35140.94} C_VEL
LIN {X 0,Y 759.907,Z 190.579,A -85,B 0,C 180,E1 35138.106,E2 35138.106} C_VEL
LIN {X 0,Y 759.919,Z 190.577,A -85,B 0,C 180,E1 35135.192,E2 35135.192} C_VEL
LIN {X 0,Y 759.911,Z 190.578,A -85,B 0,C 180,E1 35132.291,E2 35132.291} C_VEL
LIN {X 0,Y 759.904,Z 190.635,A -85,B 0,C 180,E1 35132.113,E2 35132.113} C_VEL
LIN {X 0,Y 759.914,Z 241.509,A -85,B 0,C 180,E1 35129.393,E2 35129.393} C_VEL
LIN {X 0,Y 759.875,Z 296.655,A -85,B 0,C 180,E1 35126.492,E2 35126.492} C_VEL
LIN {X 0,Y 759.873,Z 345.368,A -85,B 0,C 180,E1 35123.95,E2 35123.95} C_VEL
LIN {X 0,Y 759.905,Z 400.989,A -85,B 0,C 180,E1 35121.107,E2 35121.107} C_VEL
LIN {X 0,Y 759.874,Z 457.176,A -85,B 0,C 180,E1 35118.29,E2 35118.29} C_VEL
LIN {X 0,Y 759.867,Z 470.197,A -85,B 0,C 180,E1 35117.65,E2 35117.65} C_VEL
LIN {X 0,Y 759.915,Z 679.188,A -85,B 0,C 180,E1 35115.612,E2 35115.612} C_VEL
LIN {X 0,Y 759.914,Z 698.227,A -85,B 0,C 180,E1 35115.287,E2 35115.287} C_VEL
LIN {X 0,Y 759.916,Z 716.693,A -85,B 0,C 180,E1 35114.828,E2 35114.828} C_VEL
LIN {X 0,Y 759.892,Z 734.388,A -85,B 0,C 180,E1 35114.245,E2 35114.245} C_VEL
LIN {X 0,Y 759.918,Z 751.15,A -85,B 0,C 180,E1 35113.545,E2 35113.545} C_VEL
LIN {X 0,Y 759.917,Z 767.025,A -85,B 0,C 180,E1 35112.732,E2 35112.732} C_VEL
LIN {X 0,Y 759.916,Z 782.388,A -85,B 0,C 180,E1 35111.777,E2 35111.777} C_VEL
LIN {X 0,Y 759.918,Z 795.899,A -85,B 0,C 180,E1 35110.769,E2 35110.769} C_VEL
LIN {X 0,Y 759.918,Z 808.722,A -85,B 0,C 180,E1 35109.62,E2 35109.62} C_VEL
LIN {X 0,Y 759.913,Z 819.984,A -85,B 0,C 180,E1 35108.398,E2 35108.398} C_VEL
LIN {X 0,Y 759.919,Z 829.698,A -85,B 0,C 180,E1 35107.105,E2 35107.105} C_VEL
LIN {X 0,Y 759.911,Z 837.436,A -85,B 0,C 180,E1 35105.815,E2 35105.815} C_VEL
LIN {X 0,Y 759.91,Z 843.729,A -85,B 0,C 180,E1 35104.453,E2 35104.453} C_VEL
LIN {X 0,Y 759.916,Z 848.455,A -85,B 0,C 180,E1 35103.017,E2 35103.017} C_VEL
LIN {X 0,Y 759.909,Z 851.332,A -85,B 0,C 180,E1 35101.583,E2 35101.583} C_VEL
LIN {X 0,Y 759.911,Z 852.449,A -85,B 0,C 180,E1 35100.151,E2 35100.151} C_VEL
LIN {X 0,Y 759.915,Z 851.822,A -85,B 0,C 180,E1 35098.718,E2 35098.718} C_VEL
LIN {X 0,Y 759.911,Z 849.442,A -85,B 0,C 180,E1 35097.285,E2 35097.285} C_VEL
LIN {X 0,Y 759.915,Z 848.921,A -85,B 0,C 180,E1 35097.065,E2 35097.065} C_VEL
LIN {X 0,Y 758.934,Z 847.398,A -85,B 0,C 180,E1 35096.498,E2 35096.498} C_VEL
LIN {X 0,Y 753.637,Z 843.222,A -85,B 0,C 180,E1 35095.285,E2 35095.285} C_VEL
LIN {X 0,Y 752.012,Z 840.67,A -85,B 0,C 180,E1 35094.69,E2 35094.69} C_VEL
LIN {X 0,Y 751.92,Z 839.929,A -85,B 0,C 180,E1 35094.529,E2 35094.529} C_VEL
LIN {X 0,Y 751.924,Z 832.732,A -85,B 0,C 180,E1 35093.203,E2 35093.203} C_VEL
LIN {X 0,Y 751.931,Z 823.768,A -85,B 0,C 180,E1 35091.897,E2 35091.897} C_VEL
LIN {X 0,Y 751.951,Z 813.349,A -85,B 0,C 180,E1 35090.664,E2 35090.664} C_VEL
LIN {X 0,Y 751.972,Z 801.487,A -85,B 0,C 180,E1 35089.504,E2 35089.504} C_VEL
LIN {X 0,Y 752,Z 788.155,A -85,B 0,C 180,E1 35088.418,E2 35088.418} C_VEL
LIN {X 0,Y 752.038,Z 773.063,A -85,B 0,C 180,E1 35087.398,E2 35087.398} C_VEL
LIN {X 0,Y 752.076,Z 757.188,A -85,B 0,C 180,E1 35086.515,E2 35086.515} C_VEL
LIN {X 0,Y 752.089,Z 740.168,A -85,B 0,C 180,E1 35085.742,E2 35085.742} C_VEL
LIN {X 0,Y 752.14,Z 723.078,A -85,B 0,C 180,E1 35085.121,E2 35085.121} C_VEL
LIN {X 0,Y 752.176,Z 704.904,A -85,B 0,C 180,E1 35084.614,E2 35084.614} C_VEL
LIN {X 0,Y 752.196,Z 686.353,A -85,B 0,C 180,E1 35084.242,E2 35084.242} C_VEL
LIN {X 0,Y 752.21,Z 666.095,A -85,B 0,C 180,E1 35083.989,E2 35083.989} C_VEL
LIN {X 0,Y 752.136,Z 469.964,A -85,B 0,C 180,E1 35082.066,E2 35082.066} C_VEL
LIN {X 0,Y 752.257,Z 417.424,A -85,B 0,C 180,E1 35079.417,E2 35079.417} C_VEL
LIN {X 0,Y 752.379,Z 362.284,A -85,B 0,C 180,E1 35076.586,E2 35076.586} C_VEL
LIN {X 0,Y 752.492,Z 307.934,A -85,B 0,C 180,E1 35073.738,E2 35073.738} C_VEL
LIN {X 0,Y 752.583,Z 254.056,A -85,B 0,C 180,E1 35070.86,E2 35070.86} C_VEL
LIN {X 0,Y 752.671,Z 201.517,A -85,B 0,C 180,E1 35067.991,E2 35067.991} C_VEL
LIN {X 0,Y 752.478,Z 193.596,A -85,B 0,C 180,E1 35067.542,E2 35067.542} C_VEL
LIN {X 0,Y 751.962,Z 191.568,A -85,B 0,C 180,E1 35067.393,E2 35067.393} C_VEL
LIN {X 0,Y 751.971,Z 191.559,A -85,B 0,C 180,E1 35064.466,E2 35064.466} C_VEL
LIN {X 0,Y 751.922,Z 191.566,A -85,B 0,C 180,E1 35061.681,E2 35061.681} C_VEL
LIN {X 0,Y 751.926,Z 191.567,A -85,B 0,C 180,E1 35059.053,E2 35059.053} C_VEL
LIN {X 0,Y 751.942,Z 191.561,A -85,B 0,C 180,E1 35056.114,E2 35056.114} C_VEL
LIN {X 0,Y 751.958,Z 191.564,A -85,B 0,C 180,E1 35053.325,E2 35053.325} C_VEL
LIN {X 0,Y 751.97,Z 191.561,A -85,B 0,C 180,E1 35050.458,E2 35050.458} C_VEL
LIN {X 0,Y 751.896,Z 191.567,A -85,B 0,C 180,E1 35047.618,E2 35047.618} C_VEL
LIN {X 0,Y 751.975,Z 191.567,A -85,B 0,C 180,E1 35044.966,E2 35044.966} C_VEL
LIN {X 0,Y 751.989,Z 191.757,A -85,B 0,C 180,E1 35043.036,E2 35043.036} C_VEL
LIN {X 0,Y 752.683,Z 195.206,A -85,B 0,C 180,E1 35042.764,E2 35042.764} C_VEL
LIN {X 0,Y 752.559,Z 237.189,A -85,B 0,C 180,E1 35039.932,E2 35039.932} C_VEL
LIN {X 0,Y 752.445,Z 278.045,A -85,B 0,C 180,E1 35037.251,E2 35037.251} C_VEL
LIN {X 0,Y 752.489,Z 304.728,A -85,B 0,C 180,E1 35035.556,E2 35035.556} C_VEL
LIN {X 0,Y 752.564,Z 509.773,A -85,B 0,C 180,E1 35033.446,E2 35033.446} C_VEL
LIN {X 0,Y 752.502,Z 608.173,A -85,B 0,C 180,E1 35032.427,E2 35032.427} C_VEL
LIN {X 0,Y 752.467,Z 629.934,A -85,B 0,C 180,E1 35032.061,E2 35032.061} C_VEL
LIN {X 0,Y 752.401,Z 651.555,A -85,B 0,C 180,E1 35031.558,E2 35031.558} C_VEL
LIN {X 0,Y 752.359,Z 671.97,A -85,B 0,C 180,E1 35030.947,E2 35030.947} C_VEL
LIN {X 0,Y 752.31,Z 691.62,A -85,B 0,C 180,E1 35030.216,E2 35030.216} C_VEL
LIN {X 0,Y 752.24,Z 711.995,A -85,B 0,C 180,E1 35029.309,E2 35029.309} C_VEL
LIN {X 0,Y 752.189,Z 730.643,A -85,B 0,C 180,E1 35028.324,E2 35028.324} C_VEL
LIN {X 0,Y 752.124,Z 748.364,A -85,B 0,C 180,E1 35027.22,E2 35027.22} C_VEL
LIN {X 0,Y 752.075,Z 765.609,A -85,B 0,C 180,E1 35025.975,E2 35025.975} C_VEL
LIN {X 0,Y 752.023,Z 781.521,A -85,B 0,C 180,E1 35024.633,E2 35024.633} C_VEL
LIN {X 0,Y 751.987,Z 795.517,A -85,B 0,C 180,E1 35023.265,E2 35023.265} C_VEL
LIN {X 0,Y 751.957,Z 808.092,A -85,B 0,C 180,E1 35021.816,E2 35021.816} C_VEL
LIN {X 0,Y 751.943,Z 819.54,A -85,B 0,C 180,E1 35020.258,E2 35020.258} C_VEL
LIN {X 0,Y 751.927,Z 829.021,A -85,B 0,C 180,E1 35018.719,E2 35018.719} C_VEL
LIN {X 0,Y 751.923,Z 837.026,A -85,B 0,C 180,E1 35017.104,E2 35017.104} C_VEL
LIN {X 0,Y 751.912,Z 843.251,A -85,B 0,C 180,E1 35015.494,E2 35015.494} C_VEL
LIN {X 0,Y 751.914,Z 847.891,A -85,B 0,C 180,E1 35013.889,E2 35013.889} C_VEL
LIN {X 0,Y 751.91,Z 850.94,A -85,B 0,C 180,E1 35012.21,E2 35012.21} C_VEL
LIN {X 0,Y 751.9,Z 852.365,A -85,B 0,C 180,E1 35010.457,E2 35010.457} C_VEL
LIN {X 0,Y 751.9,Z 852.053,A -85,B 0,C 180,E1 35008.781,E2 35008.781} C_VEL
LIN {X 0,Y 751.911,Z 850.178,A -85,B 0,C 180,E1 35007.18,E2 35007.18} C_VEL
LIN {X 0,Y 751.916,Z 846.523,A -85,B 0,C 180,E1 35005.5,E2 35005.5} C_VEL
LIN {X 0,Y 751.922,Z 841.146,A -85,B 0,C 180,E1 35003.817,E2 35003.817} C_VEL
LIN {X 0,Y 751.908,Z 834.613,A -85,B 0,C 180,E1 35002.281,E2 35002.281} C_VEL
LIN {X 0,Y 751.919,Z 825.944,A -85,B 0,C 180,E1 35000.663,E2 35000.663} C_VEL
LIN {X 0,Y 751.938,Z 815.876,A -85,B 0,C 180,E1 34999.116,E2 34999.116} C_VEL
LIN {X 0,Y 751.963,Z 804.355,A -85,B 0,C 180,E1 34997.638,E2 34997.638} C_VEL
LIN {X 0,Y 751.993,Z 791.447,A -85,B 0,C 180,E1 34996.231,E2 34996.231} C_VEL
LIN {X 0,Y 752.036,Z 776.825,A -85,B 0,C 180,E1 34994.858,E2 34994.858} C_VEL
LIN {X 0,Y 752.09,Z 760.604,A -85,B 0,C 180,E1 34993.55,E2 34993.55} C_VEL
LIN {X 0,Y 752.135,Z 743.315,A -85,B 0,C 180,E1 34992.356,E2 34992.356} C_VEL
LIN {X 0,Y 752.198,Z 725.014,A -85,B 0,C 180,E1 34991.275,E2 34991.275} C_VEL
LIN {X 0,Y 752.267,Z 704.917,A -85,B 0,C 180,E1 34990.269,E2 34990.269} C_VEL
LIN {X 0,Y 752.326,Z 685.794,A -85,B 0,C 180,E1 34989.459,E2 34989.459} C_VEL
LIN {X 0,Y 752.379,Z 665.874,A -85,B 0,C 180,E1 34988.768,E2 34988.768} C_VEL
LIN {X 0,Y 752.43,Z 643.294,A -85,B 0,C 180,E1 34988.143,E2 34988.143} C_VEL
LIN {X 0,Y 752.476,Z 622.182,A -85,B 0,C 180,E1 34987.7,E2 34987.7} C_VEL
LIN {X 0,Y 752.51,Z 601.168,A -85,B 0,C 180,E1 34987.399,E2 34987.399} C_VEL
LIN {X 0,Y 752.676,Z 308.211,A -85,B 0,C 180,E1 34984.397,E2 34984.397} C_VEL
LIN {X 0,Y 752.398,Z 304.113,A -85,B 0,C 180,E1 34984.338,E2 34984.338} C_VEL
LIN {X 0,Y 752.519,Z 258.409,A -85,B 0,C 180,E1 34981.38,E2 34981.38} C_VEL
LIN {X 0,Y 752.608,Z 216.167,A -85,B 0,C 180,E1 34978.57,E2 34978.57} C_VEL
LIN {X 0,Y 752.567,Z 193.836,A -85,B 0,C 180,E1 34977.046,E2 34977.046} C_VEL
LIN {X 0,Y 751.936,Z 191.567,A -85,B 0,C 180,E1 34976.848,E2 34976.848} C_VEL
LIN {X 0,Y 751.967,Z 191.562,A -85,B 0,C 180,E1 34974.076,E2 34974.076} C_VEL
LIN {X 0,Y 751.945,Z 191.558,A -85,B 0,C 180,E1 34971.222,E2 34971.222} C_VEL
LIN {X 0,Y 751.976,Z 191.566,A -85,B 0,C 180,E1 34968.33,E2 34968.33} C_VEL
LIN {X 0,Y 751.962,Z 191.555,A -85,B 0,C 180,E1 34965.349,E2 34965.349} C_VEL
LIN {X 0,Y 751.969,Z 191.565,A -85,B 0,C 180,E1 34962.389,E2 34962.389} C_VEL
LIN {X 0,Y 751.967,Z 191.554,A -85,B 0,C 180,E1 34959.366,E2 34959.366} C_VEL
LIN {X 0,Y 751.971,Z 191.565,A -85,B 0,C 180,E1 34956.374,E2 34956.374} C_VEL
LIN {X 0,Y 751.975,Z 191.552,A -85,B 0,C 180,E1 34953.31,E2 34953.31} C_VEL
LIN {X 0,Y 751.978,Z 191.566,A -85,B 0,C 180,E1 34950.262,E2 34950.262} C_VEL
LIN {X 0,Y 751.971,Z 191.553,A -85,B 0,C 180,E1 34947.221,E2 34947.221} C_VEL
LIN {X 0,Y 751.973,Z 191.564,A -85,B 0,C 180,E1 34944.193,E2 34944.193} C_VEL
LIN {X 0,Y 751.976,Z 191.553,A -85,B 0,C 180,E1 34941.203,E2 34941.203} C_VEL
LIN {X 0,Y 751.976,Z 191.565,A -85,B 0,C 180,E1 34938.209,E2 34938.209} C_VEL
LIN {X 0,Y 751.979,Z 191.552,A -85,B 0,C 180,E1 34935.186,E2 34935.186} C_VEL
LIN {X 0,Y 751.97,Z 191.564,A -85,B 0,C 180,E1 34932.128,E2 34932.128} C_VEL
LIN {X 0,Y 751.977,Z 191.553,A -85,B 0,C 180,E1 34929.104,E2 34929.104} C_VEL
LIN {X 0,Y 751.971,Z 191.564,A -85,B 0,C 180,E1 34926.106,E2 34926.106} C_VEL
LIN {X 0,Y 751.968,Z 191.554,A -85,B 0,C 180,E1 34923.125,E2 34923.125} C_VEL
LIN {X 0,Y 751.969,Z 191.563,A -85,B 0,C 180,E1 34920.076,E2 34920.076} C_VEL
LIN {X 0,Y 751.964,Z 191.554,A -85,B 0,C 180,E1 34917.104,E2 34917.104} C_VEL
LIN {X 0,Y 751.966,Z 191.563,A -85,B 0,C 180,E1 34914.047,E2 34914.047} C_VEL
LIN {X 0,Y 751.947,Z 191.556,A -85,B 0,C 180,E1 34911.204,E2 34911.204} C_VEL
LIN {X 0,Y 751.972,Z 191.564,A -85,B 0,C 180,E1 34908.262,E2 34908.262} C_VEL
LIN {X 0,Y 751.933,Z 191.56,A -85,B 0,C 180,E1 34905.481,E2 34905.481} C_VEL
LIN {X 0,Y 751.973,Z 191.556,A -85,B 0,C 180,E1 34902.671,E2 34902.671} C_VEL
LIN {X 0,Y 751.942,Z 191.563,A -85,B 0,C 180,E1 34899.773,E2 34899.773} C_VEL
LIN {X 0,Y 751.949,Z 191.556,A -85,B 0,C 180,E1 34896.987,E2 34896.987} C_VEL
LIN {X 0,Y 751.963,Z 191.565,A -85,B 0,C 180,E1 34893.972,E2 34893.972} C_VEL
LIN {X 0,Y 751.927,Z 191.559,A -85,B 0,C 180,E1 34891.201,E2 34891.201} C_VEL
LIN {X 0,Y 751.972,Z 191.56,A -85,B 0,C 180,E1 34888.406,E2 34888.406} C_VEL
LIN {X 0,Y 751.927,Z 191.563,A -85,B 0,C 180,E1 34885.587,E2 34885.587} C_VEL
LIN {X 0,Y 751.936,Z 191.558,A -85,B 0,C 180,E1 34882.926,E2 34882.926} C_VEL
LIN {X 0,Y 751.963,Z 191.566,A -85,B 0,C 180,E1 34879.941,E2 34879.941} C_VEL
LIN {X 0,Y 751.915,Z 191.561,A -85,B 0,C 180,E1 34877.227,E2 34877.227} C_VEL
LIN {X 0,Y 751.975,Z 191.557,A -85,B 0,C 180,E1 34874.487,E2 34874.487} C_VEL
LIN {X 0,Y 751.923,Z 191.565,A -85,B 0,C 180,E1 34871.572,E2 34871.572} C_VEL
LIN {X 0,Y 751.912,Z 191.563,A -85,B 0,C 180,E1 34869.049,E2 34869.049} C_VEL
LIN {X 0,Y 751.997,Z 191.716,A -85,B 0,C 180,E1 34867.997,E2 34867.997} C_VEL
LIN {X 0,Y 753.176,Z 195.335,A -85,B 0,C 180,E1 34867.761,E2 34867.761} C_VEL
LIN {X 0,Y 753.045,Z 246.256,A -85,B 0,C 180,E1 34865.468,E2 34865.468} C_VEL
LIN {X 0,Y 753.039,Z 299.258,A -85,B 0,C 180,E1 34863.163,E2 34863.163} C_VEL
LIN {X 0,Y 753.011,Z 482.255,A -85,B 0,C 180,E1 34861.145,E2 34861.145} C_VEL
LIN {X 0,Y 752.88,Z 690.317,A -85,B 0,C 180,E1 34858.883,E2 34858.883} C_VEL
LIN {X 0,Y 752.816,Z 714.951,A -85,B 0,C 180,E1 34858.486,E2 34858.486} C_VEL
LIN {X 0,Y 752.759,Z 736.493,A -85,B 0,C 180,E1 34858.008,E2 34858.008} C_VEL
LIN {X 0,Y 752.689,Z 756.949,A -85,B 0,C 180,E1 34857.449,E2 34857.449} C_VEL
LIN {X 0,Y 752.615,Z 781.11,A -85,B 0,C 180,E1 34856.64,E2 34856.64} C_VEL
LIN {X 0,Y 752.545,Z 800.249,A -85,B 0,C 180,E1 34855.879,E2 34855.879} C_VEL
LIN {X 0,Y 752.468,Z 821.463,A -85,B 0,C 180,E1 34854.912,E2 34854.912} C_VEL
LIN {X 0,Y 752.363,Z 842.518,A -85,B 0,C 180,E1 34853.788,E2 34853.788} C_VEL
LIN {X 0,Y 752.295,Z 862.354,A -85,B 0,C 180,E1 34852.589,E2 34852.589} C_VEL
LIN {X 0,Y 752.197,Z 881.68,A -85,B 0,C 180,E1 34851.241,E2 34851.241} C_VEL
LIN {X 0,Y 752.125,Z 899.816,A -85,B 0,C 180,E1 34849.816,E2 34849.816} C_VEL
LIN {X 0,Y 752.084,Z 915.944,A -85,B 0,C 180,E1 34848.366,E2 34848.366} C_VEL
LIN {X 0,Y 752.014,Z 931.676,A -85,B 0,C 180,E1 34846.77,E2 34846.77} C_VEL
LIN {X 0,Y 751.976,Z 944.607,A -85,B 0,C 180,E1 34845.265,E2 34845.265} C_VEL
LIN {X 0,Y 751.965,Z 957.329,A -85,B 0,C 180,E1 34843.586,E2 34843.586} C_VEL
LIN {X 0,Y 751.937,Z 968.175,A -85,B 0,C 180,E1 34841.895,E2 34841.895} C_VEL
LIN {X 0,Y 751.937,Z 977.231,A -85,B 0,C 180,E1 34840.256,E2 34840.256} C_VEL
LIN {X 0,Y 751.902,Z 985.821,A -85,B 0,C 180,E1 34838.355,E2 34838.355} C_VEL
LIN {X 0,Y 751.91,Z 991.489,A -85,B 0,C 180,E1 34836.797,E2 34836.797} C_VEL
LIN {X 0,Y 751.888,Z 996.701,A -85,B 0,C 180,E1 34834.959,E2 34834.959} C_VEL
LIN {X 0,Y 751.892,Z 1000.009,A -85,B 0,C 180,E1 34833.202,E2 34833.202} C_VEL
LIN {X 0,Y 751.898,Z 1001.898,A -85,B 0,C 180,E1 34831.524,E2 34831.524} C_VEL
LIN {X 0,Y 751.885,Z 1002.395,A -85,B 0,C 180,E1 34829.619,E2 34829.619} C_VEL
LIN {X 0,Y 751.914,Z 1001.497,A -85,B 0,C 180,E1 34828.019,E2 34828.019} C_VEL
LIN {X 0,Y 751.913,Z 998.922,A -85,B 0,C 180,E1 34826.111,E2 34826.111} C_VEL
LIN {X 0,Y 751.904,Z 994.893,A -85,B 0,C 180,E1 34824.353,E2 34824.353} C_VEL
LIN {X 0,Y 751.888,Z 989.708,A -85,B 0,C 180,E1 34822.665,E2 34822.665} C_VEL
LIN {X 0,Y 751.923,Z 982.309,A -85,B 0,C 180,E1 34820.818,E2 34820.818} C_VEL
LIN {X 0,Y 751.909,Z 974.74,A -85,B 0,C 180,E1 34819.27,E2 34819.27} C_VEL
LIN {X 0,Y 751.955,Z 964.931,A -85,B 0,C 180,E1 34817.56,E2 34817.56} C_VEL
LIN {X 0,Y 751.978,Z 953.108,A -85,B 0,C 180,E1 34815.838,E2 34815.838} C_VEL
LIN {X 0,Y 752.003,Z 940.115,A -85,B 0,C 180,E1 34814.182,E2 34814.182} C_VEL
LIN {X 0,Y 752.047,Z 925.618,A -85,B 0,C 180,E1 34812.593,E2 34812.593} C_VEL
LIN {X 0,Y 752.093,Z 909.989,A -85,B 0,C 180,E1 34811.071,E2 34811.071} C_VEL
LIN {X 0,Y 752.164,Z 892.832,A -85,B 0,C 180,E1 34809.617,E2 34809.617} C_VEL
LIN {X 0,Y 752.239,Z 874.473,A -85,B 0,C 180,E1 34808.232,E2 34808.232} C_VEL
LIN {X 0,Y 752.311,Z 855.738,A -85,B 0,C 180,E1 34806.999,E2 34806.999} C_VEL
LIN {X 0,Y 752.413,Z 835.152,A -85,B 0,C 180,E1 34805.797,E2 34805.797} C_VEL
LIN {X 0,Y 752.488,Z 814.341,A -85,B 0,C 180,E1 34804.752,E2 34804.752} C_VEL
LIN {X 0,Y 752.568,Z 793.275,A -85,B 0,C 180,E1 34803.825,E2 34803.825} C_VEL
LIN {X 0,Y 752.643,Z 770.231,A -85,B 0,C 180,E1 34802.977,E2 34802.977} C_VEL
LIN {X 0,Y 752.711,Z 750.339,A -85,B 0,C 180,E1 34802.358,E2 34802.358} C_VEL
LIN {X 0,Y 752.794,Z 725.121,A -85,B 0,C 180,E1 34801.725,E2 34801.725} C_VEL
LIN {X 0,Y 752.853,Z 704.23,A -85,B 0,C 180,E1 34801.326,E2 34801.326} C_VEL
LIN {X 0,Y 752.883,Z 683.242,A -85,B 0,C 180,E1 34801.027,E2 34801.027} C_VEL
LIN {X 0,Y 753.026,Z 437.454,A -85,B 0,C 180,E1 34798.366,E2 34798.366} C_VEL
LIN {X 0,Y 753,Z 299.016,A -85,B 0,C 180,E1 34796.833,E2 34796.833} C_VEL
LIN {X 0,Y 753.055,Z 242.058,A -85,B 0,C 180,E1 34794.346,E2 34794.346} C_VEL
LIN {X 0,Y 753.192,Z 194.943,A -85,B 0,C 180,E1 34792.222,E2 34792.222} C_VEL
LIN {X 0,Y 751.954,Z 191.564,A -85,B 0,C 180,E1 34791.976,E2 34791.976} C_VEL
LIN {X 0,Y 751.93,Z 191.566,A -85,B 0,C 180,E1 34788.936,E2 34788.936} C_VEL
LIN {X 0,Y 751.937,Z 191.566,A -85,B 0,C 180,E1 34786.253,E2 34786.253} C_VEL
LIN {X 0,Y 751.965,Z 191.562,A -85,B 0,C 180,E1 34783.325,E2 34783.325} C_VEL
LIN {X 0,Y 751.927,Z 191.567,A -85,B 0,C 180,E1 34780.48,E2 34780.48} C_VEL
LIN {X 0,Y 751.97,Z 191.562,A -85,B 0,C 180,E1 34777.614,E2 34777.614} C_VEL
LIN {X 0,Y 751.926,Z 191.567,A -85,B 0,C 180,E1 34774.691,E2 34774.691} C_VEL
LIN {X 0,Y 752.003,Z 191.814,A -85,B 0,C 180,E1 34772.411,E2 34772.411} C_VEL
LIN {X 0,Y 752.705,Z 195.046,A -85,B 0,C 180,E1 34772.2,E2 34772.2} C_VEL
LIN {X 0,Y 752.544,Z 245.903,A -85,B 0,C 180,E1 34769.447,E2 34769.447} C_VEL
LIN {X 0,Y 752.472,Z 304.583,A -85,B 0,C 180,E1 34766.348,E2 34766.348} C_VEL
LIN {X 0,Y 752.372,Z 357.357,A -85,B 0,C 180,E1 34763.58,E2 34763.58} C_VEL
LIN {X 0,Y 752.253,Z 412.462,A -85,B 0,C 180,E1 34760.746,E2 34760.746} C_VEL
LIN {X 0,Y 752.142,Z 464.375,A -85,B 0,C 180,E1 34758.124,E2 34758.124} C_VEL
LIN {X 0,Y 752.211,Z 470.681,A -85,B 0,C 180,E1 34757.832,E2 34757.832} C_VEL
LIN {X 0,Y 752.205,Z 679.866,A -85,B 0,C 180,E1 34755.767,E2 34755.767} C_VEL
LIN {X 0,Y 752.179,Z 698.91,A -85,B 0,C 180,E1 34755.433,E2 34755.433} C_VEL
LIN {X 0,Y 752.151,Z 716.707,A -85,B 0,C 180,E1 34754.985,E2 34754.985} C_VEL
LIN {X 0,Y 752.094,Z 734.398,A -85,B 0,C 180,E1 34754.395,E2 34754.395} C_VEL
LIN {X 0,Y 752.083,Z 751.156,A -85,B 0,C 180,E1 34753.689,E2 34753.689} C_VEL
LIN {X 0,Y 752.047,Z 767.03,A -85,B 0,C 180,E1 34752.868,E2 34752.868} C_VEL
LIN {X 0,Y 752.014,Z 781.972,A -85,B 0,C 180,E1 34751.932,E2 34751.932} C_VEL
LIN {X 0,Y 751.983,Z 795.905,A -85,B 0,C 180,E1 34750.884,E2 34750.884} C_VEL
LIN {X 0,Y 751.959,Z 808.728,A -85,B 0,C 180,E1 34749.722,E2 34749.722} C_VEL
LIN {X 0,Y 751.939,Z 819.989,A -85,B 0,C 180,E1 34748.488,E2 34748.488} C_VEL
LIN {X 0,Y 751.93,Z 829.702,A -85,B 0,C 180,E1 34747.181,E2 34747.181} C_VEL
LIN {X 0,Y 751.919,Z 837.439,A -85,B 0,C 180,E1 34745.877,E2 34745.877} C_VEL
LIN {X 0,Y 751.912,Z 843.732,A -85,B 0,C 180,E1 34744.5,E2 34744.5} C_VEL
LIN {X 0,Y 751.916,Z 848.457,A -85,B 0,C 180,E1 34743.049,E2 34743.049} C_VEL
LIN {X 0,Y 751.91,Z 851.333,A -85,B 0,C 180,E1 34741.6,E2 34741.6} C_VEL
LIN {X 0,Y 751.911,Z 852.449,A -85,B 0,C 180,E1 34740.152,E2 34740.152} C_VEL
LIN {X 0,Y 751.915,Z 851.822,A -85,B 0,C 180,E1 34738.705,E2 34738.705} C_VEL
LIN {X 0,Y 751.911,Z 849.442,A -85,B 0,C 180,E1 34737.256,E2 34737.256} C_VEL
LIN {X 0,Y 751.913,Z 845.241,A -85,B 0,C 180,E1 34735.806,E2 34735.806} C_VEL
LIN {X 0,Y 751.92,Z 839.929,A -85,B 0,C 180,E1 34734.529,E2 34734.529} C_VEL
LIN {X 0,Y 750.931,Z 837.282,A -85,B 0,C 180,E1 34733.977,E2 34733.977} C_VEL
LIN {X 0,Y 745.826,Z 830.999,A -85,B 0,C 180,E1 34732.849,E2 34732.849} C_VEL
LIN {X 0,Y 744.047,Z 827.019,A -85,B 0,C 180,E1 34732.251,E2 34732.251} C_VEL
LIN {X 0,Y 743.951,Z 825.924,A -85,B 0,C 180,E1 34732.101,E2 34732.101} C_VEL
LIN {X 0,Y 743.984,Z 816.161,A -85,B 0,C 180,E1 34730.875,E2 34730.875} C_VEL
LIN {X 0,Y 744.022,Z 804.314,A -85,B 0,C 180,E1 34729.652,E2 34729.652} C_VEL
LIN {X 0,Y 744.075,Z 791.184,A -85,B 0,C 180,E1 34728.528,E2 34728.528} C_VEL
LIN {X 0,Y 744.139,Z 776.238,A -85,B 0,C 180,E1 34727.467,E2 34727.467} C_VEL
LIN {X 0,Y 744.21,Z 760.792,A -85,B 0,C 180,E1 34726.559,E2 34726.559} C_VEL
LIN {X 0,Y 744.268,Z 744.372,A -85,B 0,C 180,E1 34725.768,E2 34725.768} C_VEL
LIN {X 0,Y 744.343,Z 726.973,A -85,B 0,C 180,E1 34725.093,E2 34725.093} C_VEL
LIN {X 0,Y 744.425,Z 708.94,A -85,B 0,C 180,E1 34724.551,E2 34724.551} C_VEL
LIN {X 0,Y 744.47,Z 690.348,A -85,B 0,C 180,E1 34724.143,E2 34724.143} C_VEL
LIN {X 0,Y 744.511,Z 671.297,A -85,B 0,C 180,E1 34723.873,E2 34723.873} C_VEL
LIN {X 0,Y 744.485,Z 470.648,A -85,B 0,C 180,E1 34721.886,E2 34721.886} C_VEL
LIN {X 0,Y 744.625,Z 423.007,A -85,B 0,C 180,E1 34719.484,E2 34719.484} C_VEL
LIN {X 0,Y 744.817,Z 367.77,A -85,B 0,C 180,E1 34716.623,E2 34716.623} C_VEL
LIN {X 0,Y 745.023,Z 315.115,A -85,B 0,C 180,E1 34713.844,E2 34713.844} C_VEL
LIN {X 0,Y 745.23,Z 261.949,A -85,B 0,C 180,E1 34710.985,E2 34710.985} C_VEL
LIN {X 0,Y 745.483,Z 211.004,A -85,B 0,C 180,E1 34708.189,E2 34708.189} C_VEL
LIN {X 0,Y 745.406,Z 196.888,A -85,B 0,C 180,E1 34707.395,E2 34707.395} C_VEL
LIN {X 0,Y 744.033,Z 192.556,A -85,B 0,C 180,E1 34707.071,E2 34707.071} C_VEL
LIN {X 0,Y 744.026,Z 192.553,A -85,B 0,C 180,E1 34704.131,E2 34704.131} C_VEL
LIN {X 0,Y 743.972,Z 192.554,A -85,B 0,C 180,E1 34701.419,E2 34701.419} C_VEL
LIN {X 0,Y 744.042,Z 192.553,A -85,B 0,C 180,E1 34698.58,E2 34698.58} C_VEL
LIN {X 0,Y 744.001,Z 192.552,A -85,B 0,C 180,E1 34695.751,E2 34695.751} C_VEL
LIN {X 0,Y 744.008,Z 192.55,A -85,B 0,C 180,E1 34693.021,E2 34693.021} C_VEL
LIN {X 0,Y 744.038,Z 192.555,A -85,B 0,C 180,E1 34690.123,E2 34690.123} C_VEL
LIN {X 0,Y 743.96,Z 192.557,A -85,B 0,C 180,E1 34687.409,E2 34687.409} C_VEL
LIN {X 0,Y 744.033,Z 192.553,A -85,B 0,C 180,E1 34684.668,E2 34684.668} C_VEL
LIN {X 0,Y 744.058,Z 192.756,A -85,B 0,C 180,E1 34683.365,E2 34683.365} C_VEL
LIN {X 0,Y 745.472,Z 197.7,A -85,B 0,C 180,E1 34682.949,E2 34682.949} C_VEL
LIN {X 0,Y 745.224,Z 239.994,A -85,B 0,C 180,E1 34680.069,E2 34680.069} C_VEL
LIN {X 0,Y 744.994,Z 280.787,A -85,B 0,C 180,E1 34677.367,E2 34677.367} C_VEL
LIN {X 0,Y 744.954,Z 304.588,A -85,B 0,C 180,E1 34675.836,E2 34675.836} C_VEL
LIN {X 0,Y 745.451,Z 308.865,A -85,B 0,C 180,E1 34675.772,E2 34675.772} C_VEL
LIN {X 0,Y 745.108,Z 606.026,A -85,B 0,C 180,E1 34672.689,E2 34672.689} C_VEL
LIN {X 0,Y 745.032,Z 628.423,A -85,B 0,C 180,E1 34672.324,E2 34672.324} C_VEL
LIN {X 0,Y 744.911,Z 650.851,A -85,B 0,C 180,E1 34671.806,E2 34671.806} C_VEL
LIN {X 0,Y 744.834,Z 670.731,A -85,B 0,C 180,E1 34671.21,E2 34671.21} C_VEL
LIN {X 0,Y 744.711,Z 690.941,A -85,B 0,C 180,E1 34670.461,E2 34670.461} C_VEL
LIN {X 0,Y 744.589,Z 710.755,A -85,B 0,C 180,E1 34669.579,E2 34669.579} C_VEL
LIN {X 0,Y 744.477,Z 729.942,A -85,B 0,C 180,E1 34668.561,E2 34668.561} C_VEL
LIN {X 0,Y 744.344,Z 747.092,A -85,B 0,C 180,E1 34667.492,E2 34667.492} C_VEL
LIN {X 0,Y 744.238,Z 764.104,A -85,B 0,C 180,E1 34666.268,E2 34666.268} C_VEL
LIN {X 0,Y 744.149,Z 779.82,A -85,B 0,C 180,E1 34664.951,E2 34664.951} C_VEL
LIN {X 0,Y 744.08,Z 793.662,A -85,B 0,C 180,E1 34663.601,E2 34663.601} C_VEL
LIN {X 0,Y 744.023,Z 806.182,A -85,B 0,C 180,E1 34662.181,E2 34662.181} C_VEL
LIN {X 0,Y 743.968,Z 817.952,A -85,B 0,C 180,E1 34660.61,E2 34660.61} C_VEL
LIN {X 0,Y 743.938,Z 827.717,A -85,B 0,C 180,E1 34659.048,E2 34659.048} C_VEL
LIN {X 0,Y 743.914,Z 835.617,A -85,B 0,C 180,E1 34657.491,E2 34657.491} C_VEL
LIN {X 0,Y 743.913,Z 842.243,A -85,B 0,C 180,E1 34655.863,E2 34655.863} C_VEL
LIN {X 0,Y 743.918,Z 847.31,A -85,B 0,C 180,E1 34654.162,E2 34654.162} C_VEL
LIN {X 0,Y 743.912,Z 850.605,A -85,B 0,C 180,E1 34652.465,E2 34652.465} C_VEL
LIN {X 0,Y 743.913,Z 852.279,A -85,B 0,C 180,E1 34650.77,E2 34650.77} C_VEL
LIN {X 0,Y 743.912,Z 852.232,A -85,B 0,C 180,E1 34648.999,E2 34648.999} C_VEL
LIN {X 0,Y 743.913,Z 850.512,A -85,B 0,C 180,E1 34647.381,E2 34647.381} C_VEL
LIN {X 0,Y 743.917,Z 846.935,A -85,B 0,C 180,E1 34645.606,E2 34645.606} C_VEL
LIN {X 0,Y 743.924,Z 841.747,A -85,B 0,C 180,E1 34643.905,E2 34643.905} C_VEL
LIN {X 0,Y 743.916,Z 834.966,A -85,B 0,C 180,E1 34642.276,E2 34642.276} C_VEL
LIN {X 0,Y 743.937,Z 826.406,A -85,B 0,C 180,E1 34640.64,E2 34640.64} C_VEL
LIN {X 0,Y 743.975,Z 816.449,A -85,B 0,C 180,E1 34639.076,E2 34639.076} C_VEL
LIN {X 0,Y 744.019,Z 804.355,A -85,B 0,C 180,E1 34637.504,E2 34637.504} C_VEL
LIN {X 0,Y 744.08,Z 791.443,A -85,B 0,C 180,E1 34636.082,E2 34636.082} C_VEL
LIN {X 0,Y 744.166,Z 777.258,A -85,B 0,C 180,E1 34634.731,E2 34634.731} C_VEL
LIN {X 0,Y 744.266,Z 761.395,A -85,B 0,C 180,E1 34633.432,E2 34633.432} C_VEL
LIN {X 0,Y 744.357,Z 744.516,A -85,B 0,C 180,E1 34632.246,E2 34632.246} C_VEL
LIN {X 0,Y 744.485,Z 726.467,A -85,B 0,C 180,E1 34631.155,E2 34631.155} C_VEL
LIN {X 0,Y 744.621,Z 706.683,A -85,B 0,C 180,E1 34630.139,E2 34630.139} C_VEL
LIN {X 0,Y 744.729,Z 687.838,A -85,B 0,C 180,E1 34629.322,E2 34629.322} C_VEL
LIN {X 0,Y 744.846,Z 668.001,A -85,B 0,C 180,E1 34628.612,E2 34628.612} C_VEL
LIN {X 0,Y 744.956,Z 646.302,A -85,B 0,C 180,E1 34627.985,E2 34627.985} C_VEL
LIN {X 0,Y 745.044,Z 624.296,A -85,B 0,C 180,E1 34627.504,E2 34627.504} C_VEL
LIN {X 0,Y 745.114,Z 603.079,A -85,B 0,C 180,E1 34627.185,E2 34627.185} C_VEL
LIN {X 0,Y 745.454,Z 308.627,A -85,B 0,C 180,E1 34624.135,E2 34624.135} C_VEL
LIN {X 0,Y 744.892,Z 304.088,A -85,B 0,C 180,E1 34624.059,E2 34624.059} C_VEL
LIN {X 0,Y 745.133,Z 259.06,A -85,B 0,C 180,E1 34621.113,E2 34621.113} C_VEL
LIN {X 0,Y 745.348,Z 216.751,A -85,B 0,C 180,E1 34618.268,E2 34618.268} C_VEL
LIN {X 0,Y 745.365,Z 197.018,A -85,B 0,C 180,E1 34616.908,E2 34616.908} C_VEL
LIN {X 0,Y 744.02,Z 192.557,A -85,B 0,C 180,E1 34616.518,E2 34616.518} C_VEL
LIN {X 0,Y 744.024,Z 192.545,A -85,B 0,C 180,E1 34613.463,E2 34613.463} C_VEL
LIN {X 0,Y 744.013,Z 192.554,A -85,B 0,C 180,E1 34610.602,E2 34610.602} C_VEL
LIN {X 0,Y 744.03,Z 192.545,A -85,B 0,C 180,E1 34607.658,E2 34607.658} C_VEL
LIN {X 0,Y 744.002,Z 192.55,A -85,B 0,C 180,E1 34604.876,E2 34604.876} C_VEL
LIN {X 0,Y 744.028,Z 192.553,A -85,B 0,C 180,E1 34602.113,E2 34602.113} C_VEL
LIN {X 0,Y 744.024,Z 192.544,A -85,B 0,C 180,E1 34599.27,E2 34599.27} C_VEL
LIN {X 0,Y 744.035,Z 192.553,A -85,B 0,C 180,E1 34596.345,E2 34596.345} C_VEL
LIN {X 0,Y 744.033,Z 192.541,A -85,B 0,C 180,E1 34593.291,E2 34593.291} C_VEL
LIN {X 0,Y 744.039,Z 192.555,A -85,B 0,C 180,E1 34590.262,E2 34590.262} C_VEL
LIN {X 0,Y 744.033,Z 192.542,A -85,B 0,C 180,E1 34587.275,E2 34587.275} C_VEL
LIN {X 0,Y 744.035,Z 192.554,A -85,B 0,C 180,E1 34584.282,E2 34584.282} C_VEL
LIN {X 0,Y 744.037,Z 192.542,A -85,B 0,C 180,E1 34581.193,E2 34581.193} C_VEL
LIN {X 0,Y 744.033,Z 192.552,A -85,B 0,C 180,E1 34578.167,E2 34578.167} C_VEL
LIN {X 0,Y 744.035,Z 192.542,A -85,B 0,C 180,E1 34575.112,E2 34575.112} C_VEL
LIN {X 0,Y 744.029,Z 192.552,A -85,B 0,C 180,E1 34572.102,E2 34572.102} C_VEL
LIN {X 0,Y 744.037,Z 192.542,A -85,B 0,C 180,E1 34569.124,E2 34569.124} C_VEL
LIN {X 0,Y 744.03,Z 192.552,A -85,B 0,C 180,E1 34566.094,E2 34566.094} C_VEL
LIN {X 0,Y 744.032,Z 192.543,A -85,B 0,C 180,E1 34563.081,E2 34563.081} C_VEL
LIN {X 0,Y 744.03,Z 192.551,A -85,B 0,C 180,E1 34560.077,E2 34560.077} C_VEL
LIN {X 0,Y 744.021,Z 192.543,A -85,B 0,C 180,E1 34557.15,E2 34557.15} C_VEL
LIN {X 0,Y 744.032,Z 192.553,A -85,B 0,C 180,E1 34554.138,E2 34554.138} C_VEL
LIN {X 0,Y 744.004,Z 192.545,A -85,B 0,C 180,E1 34551.265,E2 34551.265} C_VEL
LIN {X 0,Y 744.029,Z 192.551,A -85,B 0,C 180,E1 34548.37,E2 34548.37} C_VEL
LIN {X 0,Y 743.996,Z 192.55,A -85,B 0,C 180,E1 34545.603,E2 34545.603} C_VEL
LIN {X 0,Y 744.037,Z 192.543,A -85,B 0,C 180,E1 34542.803,E2 34542.803} C_VEL
LIN {X 0,Y 744.005,Z 192.552,A -85,B 0,C 180,E1 34539.794,E2 34539.794} C_VEL
LIN {X 0,Y 744.011,Z 192.545,A -85,B 0,C 180,E1 34536.978,E2 34536.978} C_VEL
LIN {X 0,Y 744.02,Z 192.553,A -85,B 0,C 180,E1 34533.931,E2 34533.931} C_VEL
LIN {X 0,Y 743.991,Z 192.547,A -85,B 0,C 180,E1 34531.152,E2 34531.152} C_VEL
LIN {X 0,Y 744.034,Z 192.551,A -85,B 0,C 180,E1 34528.285,E2 34528.285} C_VEL
LIN {X 0,Y 743.984,Z 192.551,A -85,B 0,C 180,E1 34525.472,E2 34525.472} C_VEL
LIN {X 0,Y 744.012,Z 192.546,A -85,B 0,C 180,E1 34522.788,E2 34522.788} C_VEL
LIN {X 0,Y 743.998,Z 192.554,A -85,B 0,C 180,E1 34519.726,E2 34519.726} C_VEL
LIN {X 0,Y 743.982,Z 192.549,A -85,B 0,C 180,E1 34517.047,E2 34517.047} C_VEL
LIN {X 0,Y 744.037,Z 192.552,A -85,B 0,C 180,E1 34514.224,E2 34514.224} C_VEL
LIN {X 0,Y 743.975,Z 192.553,A -85,B 0,C 180,E1 34511.395,E2 34511.395} C_VEL
LIN {X 0,Y 743.992,Z 192.552,A -85,B 0,C 180,E1 34508.785,E2 34508.785} C_VEL
LIN {X 0,Y 744.057,Z 192.701,A -85,B 0,C 180,E1 34508.43,E2 34508.43} C_VEL
LIN {X 0,Y 745.441,Z 196.178,A -85,B 0,C 180,E1 34508.184,E2 34508.184} C_VEL
LIN {X 0,Y 746.508,Z 198.953,A -85,B 0,C 180,E1 34507.991,E2 34507.991} C_VEL
LIN {X 0,Y 746.231,Z 250.452,A -85,B 0,C 180,E1 34505.652,E2 34505.652} C_VEL
LIN {X 0,Y 746.107,Z 299.285,A -85,B 0,C 180,E1 34503.511,E2 34503.511} C_VEL
LIN {X 0,Y 746.45,Z 304.512,A -85,B 0,C 180,E1 34503.434,E2 34503.434} C_VEL
LIN {X 0,Y 746.056,Z 566.743,A -85,B 0,C 180,E1 34500.538,E2 34500.538} C_VEL
LIN {X 0,Y 745.863,Z 690.638,A -85,B 0,C 180,E1 34499.177,E2 34499.177} C_VEL
LIN {X 0,Y 745.738,Z 715.738,A -85,B 0,C 180,E1 34498.765,E2 34498.765} C_VEL
LIN {X 0,Y 745.629,Z 737.035,A -85,B 0,C 180,E1 34498.286,E2 34498.286} C_VEL
LIN {X 0,Y 745.494,Z 759.081,A -85,B 0,C 180,E1 34497.674,E2 34497.674} C_VEL
LIN {X 0,Y 745.323,Z 782.798,A -85,B 0,C 180,E1 34496.857,E2 34496.857} C_VEL
LIN {X 0,Y 745.177,Z 803.236,A -85,B 0,C 180,E1 34496.026,E2 34496.026} C_VEL
LIN {X 0,Y 744.963,Z 826.334,A -85,B 0,C 180,E1 34494.926,E2 34494.926} C_VEL
LIN {X 0,Y 744.817,Z 845.357,A -85,B 0,C 180,E1 34493.88,E2 34493.88} C_VEL
LIN {X 0,Y 744.621,Z 867.232,A -85,B 0,C 180,E1 34492.501,E2 34492.501} C_VEL
LIN {X 0,Y 744.486,Z 884.825,A -85,B 0,C 180,E1 34491.237,E2 34491.237} C_VEL
LIN {X 0,Y 744.329,Z 902.603,A -85,B 0,C 180,E1 34489.787,E2 34489.787} C_VEL
LIN {X 0,Y 744.248,Z 918.496,A -85,B 0,C 180,E1 34488.323,E2 34488.323} C_VEL
LIN {X 0,Y 744.132,Z 933.8,A -85,B 0,C 180,E1 34486.711,E2 34486.711} C_VEL
LIN {X 0,Y 744.053,Z 946.534,A -85,B 0,C 180,E1 34485.192,E2 34485.192} C_VEL
LIN {X 0,Y 743.994,Z 959.233,A -85,B 0,C 180,E1 34483.444,E2 34483.444} C_VEL
LIN {X 0,Y 743.968,Z 968.782,A -85,B 0,C 180,E1 34481.921,E2 34481.921} C_VEL
LIN {X 0,Y 743.952,Z 978.399,A -85,B 0,C 180,E1 34480.141,E2 34480.141} C_VEL
LIN {X 0,Y 743.91,Z 986.206,A -85,B 0,C 180,E1 34478.347,E2 34478.347} C_VEL
LIN {X 0,Y 743.909,Z 991.997,A -85,B 0,C 180,E1 34476.715,E2 34476.715} C_VEL
LIN {X 0,Y 743.902,Z 997.178,A -85,B 0,C 180,E1 34474.78,E2 34474.78} C_VEL
LIN {X 0,Y 743.89,Z 1000.122,A -85,B 0,C 180,E1 34473.159,E2 34473.159} C_VEL
LIN {X 0,Y 743.902,Z 1002.032,A -85,B 0,C 180,E1 34471.386,E2 34471.386} C_VEL
LIN {X 0,Y 743.883,Z 1002.373,A -85,B 0,C 180,E1 34469.538,E2 34469.538} C_VEL
LIN {X 0,Y 743.916,Z 1001.43,A -85,B 0,C 180,E1 34467.92,E2 34467.92} C_VEL
LIN {X 0,Y 743.916,Z 998.605,A -85,B 0,C 180,E1 34465.915,E2 34465.915} C_VEL
LIN {X 0,Y 743.919,Z 994.687,A -85,B 0,C 180,E1 34464.214,E2 34464.214} C_VEL
LIN {X 0,Y 743.893,Z 988.936,A -85,B 0,C 180,E1 34462.353,E2 34462.353} C_VEL
LIN {X 0,Y 743.929,Z 981.6,A -85,B 0,C 180,E1 34460.562,E2 34460.562} C_VEL
LIN {X 0,Y 743.926,Z 973.925,A -85,B 0,C 180,E1 34458.997,E2 34458.997} C_VEL
LIN {X 0,Y 743.978,Z 962.87,A -85,B 0,C 180,E1 34457.109,E2 34457.109} C_VEL
LIN {X 0,Y 744.04,Z 952.531,A -85,B 0,C 180,E1 34455.604,E2 34455.604} C_VEL
LIN {X 0,Y 744.114,Z 939.175,A -85,B 0,C 180,E1 34453.899,E2 34453.899} C_VEL
LIN {X 0,Y 744.189,Z 924.842,A -85,B 0,C 180,E1 34452.323,E2 34452.323} C_VEL
LIN {X 0,Y 744.313,Z 909.099,A -85,B 0,C 180,E1 34450.784,E2 34450.784} C_VEL
LIN {X 0,Y 744.42,Z 892.325,A -85,B 0,C 180,E1 34449.354,E2 34449.354} C_VEL
LIN {X 0,Y 744.581,Z 873.871,A -85,B 0,C 180,E1 34447.955,E2 34447.955} C_VEL
LIN {X 0,Y 744.718,Z 854.774,A -85,B 0,C 180,E1 34446.689,E2 34446.689} C_VEL
LIN {X 0,Y 744.932,Z 833.551,A -85,B 0,C 180,E1 34445.454,E2 34445.454} C_VEL
LIN {X 0,Y 745.075,Z 813.454,A -85,B 0,C 180,E1 34444.44,E2 34444.44} C_VEL
LIN {X 0,Y 745.289,Z 791.18,A -85,B 0,C 180,E1 34443.464,E2 34443.464} C_VEL
LIN {X 0,Y 745.407,Z 768.835,A -85,B 0,C 180,E1 34442.645,E2 34442.645} C_VEL
LIN {X 0,Y 745.561,Z 747.322,A -85,B 0,C 180,E1 34441.981,E2 34441.981} C_VEL
LIN {X 0,Y 745.712,Z 723.126,A -85,B 0,C 180,E1 34441.389,E2 34441.389} C_VEL
LIN {X 0,Y 745.811,Z 702.773,A -85,B 0,C 180,E1 34441.005,E2 34441.005} C_VEL
LIN {X 0,Y 745.891,Z 678.577,A -85,B 0,C 180,E1 34440.671,E2 34440.671} C_VEL
LIN {X 0,Y 746.202,Z 441.144,A -85,B 0,C 180,E1 34438.083,E2 34438.083} C_VEL
LIN {X 0,Y 746.303,Z 300.452,A -85,B 0,C 180,E1 34436.512,E2 34436.512} C_VEL
LIN {X 0,Y 746.003,Z 297.647,A -85,B 0,C 180,E1 34436.435,E2 34436.435} C_VEL
LIN {X 0,Y 746.291,Z 239.96,A -85,B 0,C 180,E1 34433.877,E2 34433.877} C_VEL
LIN {X 0,Y 746.493,Z 198.687,A -85,B 0,C 180,E1 34431.996,E2 34431.996} C_VEL
LIN {X 0,Y 744.077,Z 192.825,A -85,B 0,C 180,E1 34431.577,E2 34431.577} C_VEL
LIN {X 0,Y 744.039,Z 192.553,A -85,B 0,C 180,E1 34431.424,E2 34431.424} C_VEL
LIN {X 0,Y 744.001,Z 192.556,A -85,B 0,C 180,E1 34428.584,E2 34428.584} C_VEL
LIN {X 0,Y 744.014,Z 192.553,A -85,B 0,C 180,E1 34425.751,E2 34425.751} C_VEL
LIN {X 0,Y 744.012,Z 192.553,A -85,B 0,C 180,E1 34422.846,E2 34422.846} C_VEL
LIN {X 0,Y 743.983,Z 192.556,A -85,B 0,C 180,E1 34420.174,E2 34420.174} C_VEL
LIN {X 0,Y 744.027,Z 192.551,A -85,B 0,C 180,E1 34417.162,E2 34417.162} C_VEL
LIN {X 0,Y 743.984,Z 192.557,A -85,B 0,C 180,E1 34414.365,E2 34414.365} C_VEL
LIN {X 0,Y 744.038,Z 192.756,A -85,B 0,C 180,E1 34412.746,E2 34412.746} C_VEL
LIN {X 0,Y 745.545,Z 197.578,A -85,B 0,C 180,E1 34412.398,E2 34412.398} C_VEL
LIN {X 0,Y 745.188,Z 248.742,A -85,B 0,C 180,E1 34409.59,E2 34409.59} C_VEL
LIN {X 0,Y 744.994,Z 307.417,A -85,B 0,C 180,E1 34406.461,E2 34406.461} C_VEL
LIN {X 0,Y 744.851,Z 358.166,A -85,B 0,C 180,E1 34403.791,E2 34403.791} C_VEL
LIN {X 0,Y 744.628,Z 413.271,A -85,B 0,C 180,E1 34400.928,E2 34400.928} C_VEL
LIN {X 0,Y 744.433,Z 464.385,A -85,B 0,C 180,E1 34398.319,E2 34398.319} C_VEL
LIN {X 0,Y 744.488,Z 470.658,A -85,B 0,C 180,E1 34398.024,E2 34398.024} C_VEL
LIN {X 0,Y 744.501,Z 679.899,A -85,B 0,C 180,E1 34395.934,E2 34395.934} C_VEL
LIN {X 0,Y 744.452,Z 699.025,A -85,B 0,C 180,E1 34395.595,E2 34395.595} C_VEL
LIN {X 0,Y 744.396,Z 716.721,A -85,B 0,C 180,E1 34395.145,E2 34395.145} C_VEL
LIN {X 0,Y 744.305,Z 734.408,A -85,B 0,C 180,E1 34394.549,E2 34394.549} C_VEL
LIN {X 0,Y 744.258,Z 751.163,A -85,B 0,C 180,E1 34393.836,E2 34393.836} C_VEL
LIN {X 0,Y 744.185,Z 767.034,A -85,B 0,C 180,E1 34393.006,E2 34393.006} C_VEL
LIN {X 0,Y 744.115,Z 781.977,A -85,B 0,C 180,E1 34392.061,E2 34392.061} C_VEL
LIN {X 0,Y 744.052,Z 795.91,A -85,B 0,C 180,E1 34391.001,E2 34391.001} C_VEL
LIN {X 0,Y 744.004,Z 808.735,A -85,B 0,C 180,E1 34389.827,E2 34389.827} C_VEL
LIN {X 0,Y 743.967,Z 819.994,A -85,B 0,C 180,E1 34388.58,E2 34388.58} C_VEL
LIN {X 0,Y 743.941,Z 829.706,A -85,B 0,C 180,E1 34387.258,E2 34387.258} C_VEL
LIN {X 0,Y 743.927,Z 837.442,A -85,B 0,C 180,E1 34385.94,E2 34385.94} C_VEL
LIN {X 0,Y 743.914,Z 843.735,A -85,B 0,C 180,E1 34384.548,E2 34384.548} C_VEL
LIN {X 0,Y 743.915,Z 848.459,A -85,B 0,C 180,E1 34383.082,E2 34383.082} C_VEL
LIN {X 0,Y 743.91,Z 851.335,A -85,B 0,C 180,E1 34381.617,E2 34381.617} C_VEL
LIN {X 0,Y 743.912,Z 852.449,A -85,B 0,C 180,E1 34380.154,E2 34380.154} C_VEL
LIN {X 0,Y 743.915,Z 851.822,A -85,B 0,C 180,E1 34378.691,E2 34378.691} C_VEL
LIN {X 0,Y 743.911,Z 849.441,A -85,B 0,C 180,E1 34377.226,E2 34377.226} C_VEL
LIN {X 0,Y 743.916,Z 845.239,A -85,B 0,C 180,E1 34375.761,E2 34375.761} C_VEL
LIN {X 0,Y 743.922,Z 839.468,A -85,B 0,C 180,E1 34374.369,E2 34374.369} C_VEL
LIN {X 0,Y 743.938,Z 831.809,A -85,B 0,C 180,E1 34372.975,E2 34372.975} C_VEL
LIN {X 0,Y 743.951,Z 825.924,A -85,B 0,C 180,E1 34372.101,E2 34372.101} C_VEL
LIN {X 0,Y 742.947,Z 822.182,A -85,B 0,C 180,E1 34371.587,E2 34371.587} C_VEL
LIN {X 0,Y 736.999,Z 811.994,A -85,B 0,C 180,E1 34370.322,E2 34370.322} C_VEL
LIN {X 0,Y 736.061,Z 807.368,A -85,B 0,C 180,E1 34369.835,E2 34369.835} C_VEL
LIN {X 0,Y 736.147,Z 794.187,A -85,B 0,C 180,E1 34368.641,E2 34368.641} C_VEL
LIN {X 0,Y 736.239,Z 780.45,A -85,B 0,C 180,E1 34367.609,E2 34367.609} C_VEL
LIN {X 0,Y 736.345,Z 765.149,A -85,B 0,C 180,E1 34366.653,E2 34366.653} C_VEL
LIN {X 0,Y 736.456,Z 748.826,A -85,B 0,C 180,E1 34365.814,E2 34365.814} C_VEL
LIN {X 0,Y 736.543,Z 732.574,A -85,B 0,C 180,E1 34365.133,E2 34365.133} C_VEL
LIN {X 0,Y 736.667,Z 715.014,A -85,B 0,C 180,E1 34364.551,E2 34364.551} C_VEL
LIN {X 0,Y 736.748,Z 696.185,A -85,B 0,C 180,E1 34364.086,E2 34364.086} C_VEL
LIN {X 0,Y 736.815,Z 677.437,A -85,B 0,C 180,E1 34363.772,E2 34363.772} C_VEL
LIN {X 0,Y 736.875,Z 471.438,A -85,B 0,C 180,E1 34361.701,E2 34361.701} C_VEL
LIN {X 0,Y 736.706,Z 469.344,A -85,B 0,C 180,E1 34361.646,E2 34361.646} C_VEL
LIN {X 0,Y 736.999,Z 417.464,A -85,B 0,C 180,E1 34358.974,E2 34358.974} C_VEL
LIN {X 0,Y 737.322,Z 362.245,A -85,B 0,C 180,E1 34356.079,E2 34356.079} C_VEL
LIN {X 0,Y 737.639,Z 309.296,A -85,B 0,C 180,E1 34353.254,E2 34353.254} C_VEL
LIN {X 0,Y 737.969,Z 256.1,A -85,B 0,C 180,E1 34350.36,E2 34350.36} C_VEL
LIN {X 0,Y 738.306,Z 205.365,A -85,B 0,C 180,E1 34347.536,E2 34347.536} C_VEL
LIN {X 0,Y 738.149,Z 199.426,A -85,B 0,C 180,E1 34347.191,E2 34347.191} C_VEL
LIN {X 0,Y 736.097,Z 193.541,A -85,B 0,C 180,E1 34346.751,E2 34346.751} C_VEL
LIN {X 0,Y 736.091,Z 193.54,A -85,B 0,C 180,E1 34343.779,E2 34343.779} C_VEL
LIN {X 0,Y 736.047,Z 193.543,A -85,B 0,C 180,E1 34340.99,E2 34340.99} C_VEL
LIN {X 0,Y 736.041,Z 193.543,A -85,B 0,C 180,E1 34337.995,E2 34337.995} C_VEL
LIN {X 0,Y 736.098,Z 193.543,A -85,B 0,C 180,E1 34335.27,E2 34335.27} C_VEL
LIN {X 0,Y 736.095,Z 193.538,A -85,B 0,C 180,E1 34332.252,E2 34332.252} C_VEL
LIN {X 0,Y 736.025,Z 193.544,A -85,B 0,C 180,E1 34329.478,E2 34329.478} C_VEL
LIN {X 0,Y 736.094,Z 193.545,A -85,B 0,C 180,E1 34326.704,E2 34326.704} C_VEL
LIN {X 0,Y 736.07,Z 193.543,A -85,B 0,C 180,E1 34323.762,E2 34323.762} C_VEL
LIN {X 0,Y 736.099,Z 193.755,A -85,B 0,C 180,E1 34323.703,E2 34323.703} C_VEL
LIN {X 0,Y 738.265,Z 201.005,A -85,B 0,C 180,E1 34323.08,E2 34323.08} C_VEL
LIN {X 0,Y 737.884,Z 244.526,A -85,B 0,C 180,E1 34320.091,E2 34320.091} C_VEL
LIN {X 0,Y 737.524,Z 286.731,A -85,B 0,C 180,E1 34317.274,E2 34317.274} C_VEL
LIN {X 0,Y 737.486,Z 304.705,A -85,B 0,C 180,E1 34316.116,E2 34316.116} C_VEL
LIN {X 0,Y 738.245,Z 309.769,A -85,B 0,C 180,E1 34316.034,E2 34316.034} C_VEL
LIN {X 0,Y 737.722,Z 605.718,A -85,B 0,C 180,E1 34312.933,E2 34312.933} C_VEL
LIN {X 0,Y 737.611,Z 628.128,A -85,B 0,C 180,E1 34312.568,E2 34312.568} C_VEL
LIN {X 0,Y 737.451,Z 650.107,A -85,B 0,C 180,E1 34312.06,E2 34312.06} C_VEL
LIN {X 0,Y 737.311,Z 670.74,A -85,B 0,C 180,E1 34311.437,E2 34311.437} C_VEL
LIN {X 0,Y 737.125,Z 690.777,A -85,B 0,C 180,E1 34310.689,E2 34310.689} C_VEL
LIN {X 0,Y 736.946,Z 710.839,A -85,B 0,C 180,E1 34309.787,E2 34309.787} C_VEL
LIN {X 0,Y 736.764,Z 729.945,A -85,B 0,C 180,E1 34308.762,E2 34308.762} C_VEL
LIN {X 0,Y 736.568,Z 747.698,A -85,B 0,C 180,E1 34307.642,E2 34307.642} C_VEL
LIN {X 0,Y 736.398,Z 765.633,A -85,B 0,C 180,E1 34306.324,E2 34306.324} C_VEL
LIN {X 0,Y 736.255,Z 781.529,A -85,B 0,C 180,E1 34304.954,E2 34304.954} C_VEL
LIN {X 0,Y 736.161,Z 795.183,A -85,B 0,C 180,E1 34303.59,E2 34303.59} C_VEL
LIN {X 0,Y 736.072,Z 808.109,A -85,B 0,C 180,E1 34302.075,E2 34302.075} C_VEL
LIN {X 0,Y 736.001,Z 819.508,A -85,B 0,C 180,E1 34300.489,E2 34300.489} C_VEL
LIN {X 0,Y 735.958,Z 829.031,A -85,B 0,C 180,E1 34298.91,E2 34298.91} C_VEL
LIN {X 0,Y 735.929,Z 837.035,A -85,B 0,C 180,E1 34297.259,E2 34297.259} C_VEL
LIN {X 0,Y 735.915,Z 843.511,A -85,B 0,C 180,E1 34295.536,E2 34295.536} C_VEL
LIN {X 0,Y 735.914,Z 848.226,A -85,B 0,C 180,E1 34293.817,E2 34293.817} C_VEL
LIN {X 0,Y 735.913,Z 851.164,A -85,B 0,C 180,E1 34292.102,E2 34292.102} C_VEL
LIN {X 0,Y 735.9,Z 852.393,A -85,B 0,C 180,E1 34290.389,E2 34290.389} C_VEL
LIN {X 0,Y 735.897,Z 851.985,A -85,B 0,C 180,E1 34288.676,E2 34288.676} C_VEL
LIN {X 0,Y 735.902,Z 850.057,A -85,B 0,C 180,E1 34287.04,E2 34287.04} C_VEL
LIN {X 0,Y 735.909,Z 846.323,A -85,B 0,C 180,E1 34285.324,E2 34285.324} C_VEL
LIN {X 0,Y 735.923,Z 840.836,A -85,B 0,C 180,E1 34283.603,E2 34283.603} C_VEL
LIN {X 0,Y 735.938,Z 834.257,A -85,B 0,C 180,E1 34282.034,E2 34282.034} C_VEL
LIN {X 0,Y 735.962,Z 825.945,A -85,B 0,C 180,E1 34280.459,E2 34280.459} C_VEL
LIN {X 0,Y 736.015,Z 815.869,A -85,B 0,C 180,E1 34278.877,E2 34278.877} C_VEL
LIN {X 0,Y 736.084,Z 804.355,A -85,B 0,C 180,E1 34277.367,E2 34277.367} C_VEL
LIN {X 0,Y 736.171,Z 791.44,A -85,B 0,C 180,E1 34275.929,E2 34275.929} C_VEL
LIN {X 0,Y 736.309,Z 776.329,A -85,B 0,C 180,E1 34274.483,E2 34274.483} C_VEL
LIN {X 0,Y 736.462,Z 760.328,A -85,B 0,C 180,E1 34273.172,E2 34273.172} C_VEL
LIN {X 0,Y 736.609,Z 743.893,A -85,B 0,C 180,E1 34272.012,E2 34272.012} C_VEL
LIN {X 0,Y 736.785,Z 725.738,A -85,B 0,C 180,E1 34270.91,E2 34270.91} C_VEL
LIN {X 0,Y 736.991,Z 705.777,A -85,B 0,C 180,E1 34269.884,E2 34269.884} C_VEL
LIN {X 0,Y 737.168,Z 686.768,A -85,B 0,C 180,E1 34269.059,E2 34269.059} C_VEL
LIN {X 0,Y 737.336,Z 667.135,A -85,B 0,C 180,E1 34268.355,E2 34268.355} C_VEL
LIN {X 0,Y 737.509,Z 644.02,A -85,B 0,C 180,E1 34267.695,E2 34267.695} C_VEL
LIN {X 0,Y 737.632,Z 623.057,A -85,B 0,C 180,E1 34267.245,E2 34267.245} C_VEL
LIN {X 0,Y 737.732,Z 602.367,A -85,B 0,C 180,E1 34266.936,E2 34266.936} C_VEL
LIN {X 0,Y 738.247,Z 309.8,A -85,B 0,C 180,E1 34263.877,E2 34263.877} C_VEL
LIN {X 0,Y 737.404,Z 304.095,A -85,B 0,C 180,E1 34263.777,E2 34263.777} C_VEL
LIN {X 0,Y 737.753,Z 260.372,A -85,B 0,C 180,E1 34260.885,E2 34260.885} C_VEL
LIN {X 0,Y 738.089,Z 218.791,A -85,B 0,C 180,E1 34258.061,E2 34258.061} C_VEL
LIN {X 0,Y 738.056,Z 199.649,A -85,B 0,C 180,E1 34256.724,E2 34256.724} C_VEL
LIN {X 0,Y 736.094,Z 193.544,A -85,B 0,C 180,E1 34256.191,E2 34256.191} C_VEL
LIN {X 0,Y 736.069,Z 193.537,A -85,B 0,C 180,E1 34253.271,E2 34253.271} C_VEL
LIN {X 0,Y 736.092,Z 193.545,A -85,B 0,C 180,E1 34250.372,E2 34250.372} C_VEL
LIN {X 0,Y 736.08,Z 193.534,A -85,B 0,C 180,E1 34247.325,E2 34247.325} C_VEL
LIN {X 0,Y 736.092,Z 193.545,A -85,B 0,C 180,E1 34244.392,E2 34244.392} C_VEL
LIN {X 0,Y 736.086,Z 193.533,A -85,B 0,C 180,E1 34241.307,E2 34241.307} C_VEL
LIN {X 0,Y 736.09,Z 193.544,A -85,B 0,C 180,E1 34238.373,E2 34238.373} C_VEL
LIN {X 0,Y 736.09,Z 193.532,A -85,B 0,C 180,E1 34235.275,E2 34235.275} C_VEL
LIN {X 0,Y 736.095,Z 193.542,A -85,B 0,C 180,E1 34232.265,E2 34232.265} C_VEL
LIN {X 0,Y 736.097,Z 193.53,A -85,B 0,C 180,E1 34229.276,E2 34229.276} C_VEL
LIN {X 0,Y 736.095,Z 193.544,A -85,B 0,C 180,E1 34226.285,E2 34226.285} C_VEL
LIN {X 0,Y 736.095,Z 193.528,A -85,B 0,C 180,E1 34223.199,E2 34223.199} C_VEL
LIN {X 0,Y 736.095,Z 193.542,A -85,B 0,C 180,E1 34220.177,E2 34220.177} C_VEL
LIN {X 0,Y 736.097,Z 193.529,A -85,B 0,C 180,E1 34217.144,E2 34217.144} C_VEL
LIN {X 0,Y 736.091,Z 193.54,A -85,B 0,C 180,E1 34214.097,E2 34214.097} C_VEL
LIN {X 0,Y 736.097,Z 193.529,A -85,B 0,C 180,E1 34211.121,E2 34211.121} C_VEL
LIN {X 0,Y 736.093,Z 193.542,A -85,B 0,C 180,E1 34208.121,E2 34208.121} C_VEL
LIN {X 0,Y 736.092,Z 193.529,A -85,B 0,C 180,E1 34205.144,E2 34205.144} C_VEL
LIN {X 0,Y 736.092,Z 193.543,A -85,B 0,C 180,E1 34202.102,E2 34202.102} C_VEL
LIN {X 0,Y 736.094,Z 193.527,A -85,B 0,C 180,E1 34199.066,E2 34199.066} C_VEL
LIN {X 0,Y 736.085,Z 193.543,A -85,B 0,C 180,E1 34196.027,E2 34196.027} C_VEL
LIN {X 0,Y 736.085,Z 193.528,A -85,B 0,C 180,E1 34193.056,E2 34193.056} C_VEL
LIN {X 0,Y 736.083,Z 193.543,A -85,B 0,C 180,E1 34189.987,E2 34189.987} C_VEL
LIN {X 0,Y 736.079,Z 193.533,A -85,B 0,C 180,E1 34187.048,E2 34187.048} C_VEL
LIN {X 0,Y 736.083,Z 193.544,A -85,B 0,C 180,E1 34183.993,E2 34183.993} C_VEL
LIN {X 0,Y 736.064,Z 193.535,A -85,B 0,C 180,E1 34181.137,E2 34181.137} C_VEL
LIN {X 0,Y 736.095,Z 193.543,A -85,B 0,C 180,E1 34178.149,E2 34178.149} C_VEL
LIN {X 0,Y 736.05,Z 193.538,A -85,B 0,C 180,E1 34175.341,E2 34175.341} C_VEL
LIN {X 0,Y 736.094,Z 193.536,A -85,B 0,C 180,E1 34172.494,E2 34172.494} C_VEL
LIN {X 0,Y 736.053,Z 193.541,A -85,B 0,C 180,E1 34169.611,E2 34169.611} C_VEL
LIN {X 0,Y 736.067,Z 193.536,A -85,B 0,C 180,E1 34166.901,E2 34166.901} C_VEL
LIN {X 0,Y 736.066,Z 193.543,A -85,B 0,C 180,E1 34163.795,E2 34163.795} C_VEL
LIN {X 0,Y 736.045,Z 193.538,A -85,B 0,C 180,E1 34161.114,E2 34161.114} C_VEL
LIN {X 0,Y 736.097,Z 193.54,A -85,B 0,C 180,E1 34158.271,E2 34158.271} C_VEL
LIN {X 0,Y 736.042,Z 193.542,A -85,B 0,C 180,E1 34155.495,E2 34155.495} C_VEL
LIN {X 0,Y 736.049,Z 193.54,A -85,B 0,C 180,E1 34152.889,E2 34152.889} C_VEL
LIN {X 0,Y 736.078,Z 193.541,A -85,B 0,C 180,E1 34149.87,E2 34149.87} C_VEL
LIN {X 0,Y 736.048,Z 193.566,A -85,B 0,C 180,E1 34148.886,E2 34148.886} C_VEL
LIN {X 0,Y 737.361,Z 197.003,A -85,B 0,C 180,E1 34148.64,E2 34148.64} C_VEL
LIN {X 0,Y 739.844,Z 202.205,A -85,B 0,C 180,E1 34148.242,E2 34148.242} C_VEL
LIN {X 0,Y 739.438,Z 252.549,A -85,B 0,C 180,E1 34145.935,E2 34145.935} C_VEL
LIN {X 0,Y 739.213,Z 299.377,A -85,B 0,C 180,E1 34143.864,E2 34143.864} C_VEL
LIN {X 0,Y 739.767,Z 304.649,A -85,B 0,C 180,E1 34143.775,E2 34143.775} C_VEL
LIN {X 0,Y 739.162,Z 566.234,A -85,B 0,C 180,E1 34140.86,E2 34140.86} C_VEL
LIN {X 0,Y 738.866,Z 690.746,A -85,B 0,C 180,E1 34139.479,E2 34139.479} C_VEL
LIN {X 0,Y 738.682,Z 715.989,A -85,B 0,C 180,E1 34139.061,E2 34139.061} C_VEL
LIN {X 0,Y 738.517,Z 737.469,A -85,B 0,C 180,E1 34138.573,E2 34138.573} C_VEL
LIN {X 0,Y 738.315,Z 760.62,A -85,B 0,C 180,E1 34137.92,E2 34137.92} C_VEL
LIN {X 0,Y 738.046,Z 783.535,A -85,B 0,C 180,E1 34137.115,E2 34137.115} C_VEL
LIN {X 0,Y 737.827,Z 804.234,A -85,B 0,C 180,E1 34136.261,E2 34136.261} C_VEL
LIN {X 0,Y 737.502,Z 827.14,A -85,B 0,C 180,E1 34135.153,E2 34135.153} C_VEL
LIN {X 0,Y 737.279,Z 846.887,A -85,B 0,C 180,E1 34134.05,E2 34134.05} C_VEL
LIN {X 0,Y 736.994,Z 867.234,A -85,B 0,C 180,E1 34132.747,E2 34132.747} C_VEL
LIN {X 0,Y 736.79,Z 885.106,A -85,B 0,C 180,E1 34131.449,E2 34131.449} C_VEL
LIN {X 0,Y 736.562,Z 902.604,A -85,B 0,C 180,E1 34130.004,E2 34130.004} C_VEL
LIN {X 0,Y 736.424,Z 918.494,A -85,B 0,C 180,E1 34128.525,E2 34128.525} C_VEL
LIN {X 0,Y 736.241,Z 933.802,A -85,B 0,C 180,E1 34126.896,E2 34126.896} C_VEL
LIN {X 0,Y 736.14,Z 946.535,A -85,B 0,C 180,E1 34125.359,E2 34125.359} C_VEL
LIN {X 0,Y 736.044,Z 959.754,A -85,B 0,C 180,E1 34123.512,E2 34123.512} C_VEL
LIN {X 0,Y 736,Z 969.102,A -85,B 0,C 180,E1 34121.997,E2 34121.997} C_VEL
LIN {X 0,Y 735.967,Z 978.76,A -85,B 0,C 180,E1 34120.173,E2 34120.173} C_VEL
LIN {X 0,Y 735.912,Z 986.207,A -85,B 0,C 180,E1 34118.438,E2 34118.438} C_VEL
LIN {X 0,Y 735.917,Z 991.998,A -85,B 0,C 180,E1 34116.789,E2 34116.789} C_VEL
LIN {X 0,Y 735.898,Z 997.178,A -85,B 0,C 180,E1 34114.832,E2 34114.832} C_VEL
LIN {X 0,Y 735.892,Z 1000.122,A -85,B 0,C 180,E1 34113.193,E2 34113.193} C_VEL
LIN {X 0,Y 735.905,Z 1002.099,A -85,B 0,C 180,E1 34111.323,E2 34111.323} C_VEL
LIN {X 0,Y 735.881,Z 1002.351,A -85,B 0,C 180,E1 34109.455,E2 34109.455} C_VEL
LIN {X 0,Y 735.917,Z 1001.297,A -85,B 0,C 180,E1 34107.742,E2 34107.742} C_VEL
LIN {X 0,Y 735.914,Z 998.431,A -85,B 0,C 180,E1 34105.785,E2 34105.785} C_VEL
LIN {X 0,Y 735.923,Z 994.481,A -85,B 0,C 180,E1 34104.073,E2 34104.073} C_VEL
LIN {X 0,Y 735.907,Z 988.636,A -85,B 0,C 180,E1 34102.191,E2 34102.191} C_VEL
LIN {X 0,Y 735.937,Z 981.601,A -85,B 0,C 180,E1 34100.459,E2 34100.459} C_VEL
LIN {X 0,Y 735.951,Z 973.926,A -85,B 0,C 180,E1 34098.876,E2 34098.876} C_VEL
LIN {X 0,Y 736.02,Z 962.872,A -85,B 0,C 180,E1 34096.967,E2 34096.967} C_VEL
LIN {X 0,Y 736.106,Z 952.533,A -85,B 0,C 180,E1 34095.446,E2 34095.446} C_VEL
LIN {X 0,Y 736.223,Z 939.445,A -85,B 0,C 180,E1 34093.753,E2 34093.753} C_VEL
LIN {X 0,Y 736.329,Z 924.844,A -85,B 0,C 180,E1 34092.128,E2 34092.128} C_VEL
LIN {X 0,Y 736.525,Z 909.098,A -85,B 0,C 180,E1 34090.573,E2 34090.573} C_VEL
LIN {X 0,Y 736.688,Z 892.324,A -85,B 0,C 180,E1 34089.128,E2 34089.128} C_VEL
LIN {X 0,Y 736.935,Z 873.997,A -85,B 0,C 180,E1 34087.722,E2 34087.722} C_VEL
LIN {X 0,Y 737.141,Z 855.082,A -85,B 0,C 180,E1 34086.455,E2 34086.455} C_VEL
LIN {X 0,Y 737.455,Z 834.357,A -85,B 0,C 180,E1 34085.231,E2 34085.231} C_VEL
LIN {X 0,Y 737.671,Z 814.349,A -85,B 0,C 180,E1 34084.208,E2 34084.208} C_VEL
LIN {X 0,Y 737.994,Z 791.916,A -85,B 0,C 180,E1 34083.21,E2 34083.21} C_VEL
LIN {X 0,Y 738.186,Z 769.577,A -85,B 0,C 180,E1 34082.38,E2 34082.38} C_VEL
LIN {X 0,Y 738.413,Z 748.132,A -85,B 0,C 180,E1 34081.71,E2 34081.71} C_VEL
LIN {X 0,Y 738.644,Z 723.518,A -85,B 0,C 180,E1 34081.098,E2 34081.098} C_VEL
LIN {X 0,Y 738.787,Z 702.774,A -85,B 0,C 180,E1 34080.702,E2 34080.702} C_VEL
LIN {X 0,Y 738.912,Z 678.196,A -85,B 0,C 180,E1 34080.363,E2 34080.363} C_VEL
LIN {X 0,Y 739.404,Z 441.272,A -85,B 0,C 180,E1 34077.756,E2 34077.756} C_VEL
LIN {X 0,Y 739.616,Z 301.831,A -85,B 0,C 180,E1 34076.185,E2 34076.185} C_VEL
LIN {X 0,Y 739.094,Z 298.171,A -85,B 0,C 180,E1 34076.102,E2 34076.102} C_VEL
LIN {X 0,Y 739.553,Z 239.96,A -85,B 0,C 180,E1 34073.495,E2 34073.495} C_VEL
LIN {X 0,Y 739.783,Z 202.044,A -85,B 0,C 180,E1 34071.747,E2 34071.747} C_VEL
LIN {X 0,Y 736.248,Z 194.372,A -85,B 0,C 180,E1 34071.165,E2 34071.165} C_VEL
LIN {X 0,Y 736.098,Z 193.545,A -85,B 0,C 180,E1 34071.11,E2 34071.11} C_VEL
LIN {X 0,Y 736.098,Z 193.544,A -85,B 0,C 180,E1 34068.167,E2 34068.167} C_VEL
LIN {X 0,Y 736.094,Z 193.545,A -85,B 0,C 180,E1 34065.27,E2 34065.27} C_VEL
LIN {X 0,Y 736.094,Z 193.544,A -85,B 0,C 180,E1 34062.357,E2 34062.357} C_VEL
LIN {X 0,Y 736.1,Z 193.544,A -85,B 0,C 180,E1 34059.473,E2 34059.473} C_VEL
LIN {X 0,Y 736.087,Z 193.545,A -85,B 0,C 180,E1 34056.511,E2 34056.511} C_VEL
LIN {X 0,Y 736.101,Z 193.544,A -85,B 0,C 180,E1 34053.563,E2 34053.563} C_VEL
LIN {X 0,Y 736.114,Z 193.791,A -85,B 0,C 180,E1 34053.097,E2 34053.097} C_VEL
LIN {X 0,Y 738.426,Z 200.857,A -85,B 0,C 180,E1 34052.565,E2 34052.565} C_VEL
LIN {X 0,Y 737.861,Z 251.699,A -85,B 0,C 180,E1 34049.734,E2 34049.734} C_VEL
LIN {X 0,Y 737.516,Z 310.25,A -85,B 0,C 180,E1 34046.577,E2 34046.577} C_VEL
LIN {X 0,Y 737.327,Z 364.464,A -85,B 0,C 180,E1 34043.713,E2 34043.713} C_VEL
LIN {X 0,Y 736.992,Z 419.67,A -85,B 0,C 180,E1 34040.822,E2 34040.822} C_VEL
LIN {X 0,Y 736.751,Z 470.465,A -85,B 0,C 180,E1 34038.222,E2 34038.222} C_VEL
LIN {X 0,Y 737.012,Z 488.726,A -85,B 0,C 180,E1 34038.032,E2 34038.032} C_VEL
LIN {X 0,Y 736.806,Z 679.936,A -85,B 0,C 180,E1 34036.105,E2 34036.105} C_VEL
LIN {X 0,Y 736.732,Z 698.968,A -85,B 0,C 180,E1 34035.765,E2 34035.765} C_VEL
LIN {X 0,Y 736.649,Z 716.735,A -85,B 0,C 180,E1 34035.308,E2 34035.308} C_VEL
LIN {X 0,Y 736.523,Z 734.417,A -85,B 0,C 180,E1 34034.707,E2 34034.707} C_VEL
LIN {X 0,Y 736.439,Z 751.17,A -85,B 0,C 180,E1 34033.986,E2 34033.986} C_VEL
LIN {X 0,Y 736.329,Z 766.972,A -85,B 0,C 180,E1 34033.151,E2 34033.151} C_VEL
LIN {X 0,Y 736.223,Z 781.982,A -85,B 0,C 180,E1 34032.192,E2 34032.192} C_VEL
LIN {X 0,Y 736.125,Z 795.916,A -85,B 0,C 180,E1 34031.121,E2 34031.121} C_VEL
LIN {X 0,Y 736.049,Z 808.741,A -85,B 0,C 180,E1 34029.935,E2 34029.935} C_VEL
LIN {X 0,Y 735.996,Z 819.999,A -85,B 0,C 180,E1 34028.673,E2 34028.673} C_VEL
LIN {X 0,Y 735.954,Z 829.711,A -85,B 0,C 180,E1 34027.337,E2 34027.337} C_VEL
LIN {X 0,Y 735.933,Z 837.547,A -85,B 0,C 180,E1 34025.985,E2 34025.985} C_VEL
LIN {X 0,Y 735.917,Z 843.738,A -85,B 0,C 180,E1 34024.598,E2 34024.598} C_VEL
LIN {X 0,Y 735.915,Z 848.461,A -85,B 0,C 180,E1 34023.115,E2 34023.115} C_VEL
LIN {X 0,Y 735.911,Z 851.337,A -85,B 0,C 180,E1 34021.635,E2 34021.635} C_VEL
LIN {X 0,Y 735.912,Z 852.449,A -85,B 0,C 180,E1 34020.156,E2 34020.156} C_VEL
LIN {X 0,Y 735.914,Z 851.821,A -85,B 0,C 180,E1 34018.676,E2 34018.676} C_VEL
LIN {X 0,Y 735.912,Z 849.439,A -85,B 0,C 180,E1 34017.196,E2 34017.196} C_VEL
LIN {X 0,Y 735.919,Z 845.237,A -85,B 0,C 180,E1 34015.714,E2 34015.714} C_VEL
LIN {X 0,Y 735.926,Z 839.466,A -85,B 0,C 180,E1 34014.308,E2 34014.308} C_VEL
LIN {X 0,Y 735.954,Z 831.807,A -85,B 0,C 180,E1 34012.898,E2 34012.898} C_VEL
LIN {X 0,Y 735.986,Z 822.611,A -85,B 0,C 180,E1 34011.563,E2 34011.563} C_VEL
LIN {X 0,Y 736.04,Z 811.927,A -85,B 0,C 180,E1 34010.302,E2 34010.302} C_VEL
LIN {X 0,Y 736.061,Z 807.368,A -85,B 0,C 180,E1 34009.835,E2 34009.835} C_VEL
LIN {X 0,Y 735.127,Z 802.66,A -85,B 0,C 180,E1 34009.36,E2 34009.36} C_VEL
LIN {X 0,Y 729.255,Z 790.206,A -85,B 0,C 180,E1 34008.209,E2 34008.209} C_VEL
LIN {X 0,Y 728.304,Z 784.724,A -85,B 0,C 180,E1 34007.782,E2 34007.782} C_VEL
LIN {X 0,Y 728.445,Z 769.201,A -85,B 0,C 180,E1 34006.748,E2 34006.748} C_VEL
LIN {X 0,Y 728.599,Z 752.979,A -85,B 0,C 180,E1 34005.861,E2 34005.861} C_VEL
LIN {X 0,Y 728.729,Z 735.644,A -85,B 0,C 180,E1 34005.092,E2 34005.092} C_VEL
LIN {X 0,Y 728.892,Z 718.299,A -85,B 0,C 180,E1 34004.484,E2 34004.484} C_VEL
LIN {X 0,Y 729.006,Z 699.867,A -85,B 0,C 180,E1 34003.994,E2 34003.994} C_VEL
LIN {X 0,Y 729.105,Z 681.174,A -85,B 0,C 180,E1 34003.649,E2 34003.649} C_VEL
LIN {X 0,Y 729.162,Z 642.014,A -85,B 0,C 180,E1 34003.228,E2 34003.228} C_VEL
LIN {X 0,Y 729.244,Z 472.056,A -85,B 0,C 180,E1 34001.509,E2 34001.509} C_VEL
LIN {X 0,Y 729.002,Z 469.734,A -85,B 0,C 180,E1 34001.466,E2 34001.466} C_VEL
LIN {X 0,Y 729.384,Z 418.134,A -85,B 0,C 180,E1 33998.779,E2 33998.779} C_VEL
LIN {X 0,Y 729.793,Z 363.729,A -85,B 0,C 180,E1 33995.902,E2 33995.902} C_VEL
LIN {X 0,Y 730.225,Z 310.78,A -85,B 0,C 180,E1 33993.048,E2 33993.048} C_VEL
LIN {X 0,Y 730.682,Z 257.539,A -85,B 0,C 180,E1 33990.125,E2 33990.125} C_VEL
LIN {X 0,Y 731.155,Z 206.399,A -85,B 0,C 180,E1 33987.251,E2 33987.251} C_VEL
LIN {X 0,Y 731.053,Z 202.8,A -85,B 0,C 180,E1 33987.039,E2 33987.039} C_VEL
LIN {X 0,Y 728.145,Z 194.532,A -85,B 0,C 180,E1 33986.399,E2 33986.399} C_VEL
LIN {X 0,Y 728.129,Z 194.531,A -85,B 0,C 180,E1 33983.515,E2 33983.515} C_VEL
LIN {X 0,Y 728.137,Z 194.532,A -85,B 0,C 180,E1 33980.724,E2 33980.724} C_VEL
LIN {X 0,Y 728.098,Z 194.532,A -85,B 0,C 180,E1 33977.866,E2 33977.866} C_VEL
LIN {X 0,Y 728.153,Z 194.531,A -85,B 0,C 180,E1 33975.104,E2 33975.104} C_VEL
LIN {X 0,Y 728.154,Z 194.529,A -85,B 0,C 180,E1 33972.139,E2 33972.139} C_VEL
LIN {X 0,Y 728.083,Z 194.533,A -85,B 0,C 180,E1 33969.381,E2 33969.381} C_VEL
LIN {X 0,Y 728.161,Z 194.533,A -85,B 0,C 180,E1 33966.553,E2 33966.553} C_VEL
LIN {X 0,Y 728.144,Z 194.584,A -85,B 0,C 180,E1 33964.048,E2 33964.048} C_VEL
LIN {X 0,Y 731.081,Z 203.706,A -85,B 0,C 180,E1 33963.26,E2 33963.26} C_VEL
LIN {X 0,Y 730.554,Z 247.173,A -85,B 0,C 180,E1 33960.243,E2 33960.243} C_VEL
LIN {X 0,Y 730.071,Z 290.037,A -85,B 0,C 180,E1 33957.355,E2 33957.355} C_VEL
LIN {X 0,Y 730.002,Z 304.646,A -85,B 0,C 180,E1 33956.406,E2 33956.406} C_VEL
LIN {X 0,Y 731.053,Z 311.118,A -85,B 0,C 180,E1 33956.295,E2 33956.295} C_VEL
LIN {X 0,Y 730.351,Z 605.307,A -85,B 0,C 180,E1 33953.183,E2 33953.183} C_VEL
LIN {X 0,Y 730.203,Z 627.683,A -85,B 0,C 180,E1 33952.82,E2 33952.82} C_VEL
LIN {X 0,Y 729.999,Z 650.119,A -85,B 0,C 180,E1 33952.297,E2 33952.297} C_VEL
LIN {X 0,Y 729.8,Z 670.734,A -85,B 0,C 180,E1 33951.669,E2 33951.669} C_VEL
LIN {X 0,Y 729.555,Z 690.687,A -85,B 0,C 180,E1 33950.918,E2 33950.918} C_VEL
LIN {X 0,Y 729.297,Z 711.654,A -85,B 0,C 180,E1 33949.961,E2 33949.961} C_VEL
LIN {X 0,Y 729.049,Z 730.631,A -85,B 0,C 180,E1 33948.927,E2 33948.927} C_VEL
LIN {X 0,Y 728.799,Z 748.01,A -85,B 0,C 180,E1 33947.815,E2 33947.815} C_VEL
LIN {X 0,Y 728.575,Z 765.645,A -85,B 0,C 180,E1 33946.504,E2 33946.504} C_VEL
LIN {X 0,Y 728.381,Z 781.531,A -85,B 0,C 180,E1 33945.119,E2 33945.119} C_VEL
LIN {X 0,Y 728.245,Z 795.18,A -85,B 0,C 180,E1 33943.741,E2 33943.741} C_VEL
LIN {X 0,Y 728.128,Z 808.117,A -85,B 0,C 180,E1 33942.209,E2 33942.209} C_VEL
LIN {X 0,Y 728.028,Z 819.511,A -85,B 0,C 180,E1 33940.605,E2 33940.605} C_VEL
LIN {X 0,Y 727.971,Z 828.845,A -85,B 0,C 180,E1 33939.042,E2 33939.042} C_VEL
LIN {X 0,Y 727.933,Z 836.92,A -85,B 0,C 180,E1 33937.366,E2 33937.366} C_VEL
LIN {X 0,Y 727.914,Z 843.261,A -85,B 0,C 180,E1 33935.676,E2 33935.676} C_VEL
LIN {X 0,Y 727.918,Z 847.875,A -85,B 0,C 180,E1 33934.017,E2 33934.017} C_VEL
LIN {X 0,Y 727.91,Z 850.83,A -85,B 0,C 180,E1 33932.362,E2 33932.362} C_VEL
LIN {X 0,Y 727.903,Z 852.352,A -85,B 0,C 180,E1 33930.551,E2 33930.551} C_VEL
LIN {X 0,Y 727.902,Z 852.106,A -85,B 0,C 180,E1 33928.819,E2 33928.819} C_VEL
LIN {X 0,Y 727.909,Z 850.288,A -85,B 0,C 180,E1 33927.166,E2 33927.166} C_VEL
LIN {X 0,Y 727.916,Z 846.735,A -85,B 0,C 180,E1 33925.43,E2 33925.43} C_VEL
LIN {X 0,Y 727.932,Z 841.437,A -85,B 0,C 180,E1 33923.691,E2 33923.691} C_VEL
LIN {X 0,Y 727.947,Z 834.613,A -85,B 0,C 180,E1 33922.026,E2 33922.026} C_VEL
LIN {X 0,Y 727.987,Z 825.946,A -85,B 0,C 180,E1 33920.354,E2 33920.354} C_VEL
LIN {X 0,Y 728.064,Z 815.288,A -85,B 0,C 180,E1 33918.674,E2 33918.674} C_VEL
LIN {X 0,Y 728.162,Z 803.686,A -85,B 0,C 180,E1 33917.147,E2 33917.147} C_VEL
LIN {X 0,Y 728.281,Z 790.661,A -85,B 0,C 180,E1 33915.692,E2 33915.692} C_VEL
LIN {X 0,Y 728.457,Z 775.036,A -85,B 0,C 180,E1 33914.198,E2 33914.198} C_VEL
LIN {X 0,Y 728.66,Z 758.929,A -85,B 0,C 180,E1 33912.882,E2 33912.882} C_VEL
LIN {X 0,Y 728.895,Z 742.043,A -85,B 0,C 180,E1 33911.691,E2 33911.691} C_VEL
LIN {X 0,Y 729.168,Z 722.09,A -85,B 0,C 180,E1 33910.494,E2 33910.494} C_VEL
LIN {X 0,Y 729.388,Z 703.091,A -85,B 0,C 180,E1 33909.539,E2 33909.539} C_VEL
LIN {X 0,Y 729.656,Z 683.618,A -85,B 0,C 180,E1 33908.707,E2 33908.707} C_VEL
LIN {X 0,Y 729.908,Z 661.286,A -85,B 0,C 180,E1 33907.933,E2 33907.933} C_VEL
LIN {X 0,Y 730.093,Z 640.176,A -85,B 0,C 180,E1 33907.363,E2 33907.363} C_VEL
LIN {X 0,Y 730.285,Z 617.845,A -85,B 0,C 180,E1 33906.911,E2 33906.911} C_VEL
LIN {X 0,Y 730.4,Z 592.796,A -85,B 0,C 180,E1 33906.58,E2 33906.58} C_VEL
LIN {X 0,Y 731.059,Z 309.801,A -85,B 0,C 180,E1 33903.601,E2 33903.601} C_VEL
LIN {X 0,Y 729.935,Z 303.922,A -85,B 0,C 180,E1 33903.476,E2 33903.476} C_VEL
LIN {X 0,Y 730.388,Z 261.023,A -85,B 0,C 180,E1 33900.608,E2 33900.608} C_VEL
LIN {X 0,Y 730.864,Z 219.442,A -85,B 0,C 180,E1 33897.754,E2 33897.754} C_VEL
LIN {X 0,Y 730.869,Z 202.718,A -85,B 0,C 180,E1 33896.568,E2 33896.568} C_VEL
LIN {X 0,Y 728.154,Z 194.53,A -85,B 0,C 180,E1 33895.831,E2 33895.831} C_VEL
LIN {X 0,Y 728.122,Z 194.529,A -85,B 0,C 180,E1 33893.024,E2 33893.024} C_VEL
LIN {X 0,Y 728.157,Z 194.532,A -85,B 0,C 180,E1 33890.215,E2 33890.215} C_VEL
LIN {X 0,Y 728.138,Z 194.524,A -85,B 0,C 180,E1 33887.28,E2 33887.28} C_VEL
LIN {X 0,Y 728.156,Z 194.532,A -85,B 0,C 180,E1 33884.322,E2 33884.322} C_VEL
LIN {X 0,Y 728.148,Z 194.522,A -85,B 0,C 180,E1 33881.311,E2 33881.311} C_VEL
LIN {X 0,Y 728.151,Z 194.534,A -85,B 0,C 180,E1 33878.363,E2 33878.363} C_VEL
LIN {X 0,Y 728.155,Z 194.521,A -85,B 0,C 180,E1 33875.318,E2 33875.318} C_VEL
LIN {X 0,Y 728.156,Z 194.53,A -85,B 0,C 180,E1 33872.288,E2 33872.288} C_VEL
LIN {X 0,Y 728.158,Z 194.519,A -85,B 0,C 180,E1 33869.265,E2 33869.265} C_VEL
LIN {X 0,Y 728.155,Z 194.534,A -85,B 0,C 180,E1 33866.242,E2 33866.242} C_VEL
LIN {X 0,Y 728.157,Z 194.516,A -85,B 0,C 180,E1 33863.21,E2 33863.21} C_VEL
LIN {X 0,Y 728.155,Z 194.53,A -85,B 0,C 180,E1 33860.162,E2 33860.162} C_VEL
LIN {X 0,Y 728.156,Z 194.517,A -85,B 0,C 180,E1 33857.112,E2 33857.112} C_VEL
LIN {X 0,Y 728.156,Z 194.529,A -85,B 0,C 180,E1 33854.148,E2 33854.148} C_VEL
LIN {X 0,Y 728.157,Z 194.518,A -85,B 0,C 180,E1 33851.084,E2 33851.084} C_VEL
LIN {X 0,Y 728.148,Z 194.529,A -85,B 0,C 180,E1 33848.052,E2 33848.052} C_VEL
LIN {X 0,Y 728.155,Z 194.517,A -85,B 0,C 180,E1 33845.042,E2 33845.042} C_VEL
LIN {X 0,Y 728.148,Z 194.531,A -85,B 0,C 180,E1 33842.046,E2 33842.046} C_VEL
LIN {X 0,Y 728.155,Z 194.515,A -85,B 0,C 180,E1 33839.056,E2 33839.056} C_VEL
LIN {X 0,Y 728.143,Z 194.531,A -85,B 0,C 180,E1 33835.984,E2 33835.984} C_VEL
LIN {X 0,Y 728.147,Z 194.516,A -85,B 0,C 180,E1 33833.059,E2 33833.059} C_VEL
LIN {X 0,Y 728.141,Z 194.531,A -85,B 0,C 180,E1 33829.956,E2 33829.956} C_VEL
LIN {X 0,Y 728.139,Z 194.522,A -85,B 0,C 180,E1 33827.066,E2 33827.066} C_VEL
LIN {X 0,Y 728.142,Z 194.532,A -85,B 0,C 180,E1 33823.977,E2 33823.977} C_VEL
LIN {X 0,Y 728.128,Z 194.523,A -85,B 0,C 180,E1 33821.113,E2 33821.113} C_VEL
LIN {X 0,Y 728.155,Z 194.533,A -85,B 0,C 180,E1 33818.068,E2 33818.068} C_VEL
LIN {X 0,Y 728.114,Z 194.526,A -85,B 0,C 180,E1 33815.238,E2 33815.238} C_VEL
LIN {X 0,Y 728.154,Z 194.527,A -85,B 0,C 180,E1 33812.338,E2 33812.338} C_VEL
LIN {X 0,Y 728.111,Z 194.53,A -85,B 0,C 180,E1 33809.553,E2 33809.553} C_VEL
LIN {X 0,Y 728.146,Z 194.524,A -85,B 0,C 180,E1 33806.749,E2 33806.749} C_VEL
LIN {X 0,Y 728.12,Z 194.531,A -85,B 0,C 180,E1 33803.71,E2 33803.71} C_VEL
LIN {X 0,Y 728.111,Z 194.527,A -85,B 0,C 180,E1 33801.011,E2 33801.011} C_VEL
LIN {X 0,Y 728.154,Z 194.532,A -85,B 0,C 180,E1 33798.03,E2 33798.03} C_VEL
LIN {X 0,Y 728.098,Z 194.53,A -85,B 0,C 180,E1 33795.321,E2 33795.321} C_VEL
LIN {X 0,Y 728.142,Z 194.528,A -85,B 0,C 180,E1 33792.605,E2 33792.605} C_VEL
LIN {X 0,Y 728.107,Z 194.53,A -85,B 0,C 180,E1 33789.583,E2 33789.583} C_VEL
LIN {X 0,Y 728.128,Z 194.767,A -85,B 0,C 180,E1 33789.332,E2 33789.332} C_VEL
LIN {X 0,Y 729.397,Z 198.009,A -85,B 0,C 180,E1 33789.094,E2 33789.094} C_VEL
LIN {X 0,Y 733.184,Z 205.799,A -85,B 0,C 180,E1 33788.482,E2 33788.482} C_VEL
LIN {X 0,Y 732.67,Z 253.703,A -85,B 0,C 180,E1 33786.266,E2 33786.266} C_VEL
LIN {X 0,Y 732.316,Z 299.265,A -85,B 0,C 180,E1 33784.229,E2 33784.229} C_VEL
LIN {X 0,Y 733.106,Z 305.86,A -85,B 0,C 180,E1 33784.11,E2 33784.11} C_VEL
LIN {X 0,Y 732.282,Z 568.349,A -85,B 0,C 180,E1 33781.158,E2 33781.158} C_VEL
LIN {X 0,Y 731.89,Z 690.853,A -85,B 0,C 180,E1 33779.787,E2 33779.787} C_VEL
LIN {X 0,Y 731.647,Z 716.249,A -85,B 0,C 180,E1 33779.362,E2 33779.362} C_VEL
LIN {X 0,Y 731.424,Z 737.796,A -85,B 0,C 180,E1 33778.867,E2 33778.867} C_VEL
LIN {X 0,Y 731.146,Z 761.29,A -85,B 0,C 180,E1 33778.196,E2 33778.196} C_VEL
LIN {X 0,Y 730.784,Z 784.275,A -85,B 0,C 180,E1 33777.378,E2 33777.378} C_VEL
LIN {X 0,Y 730.482,Z 806.069,A -85,B 0,C 180,E1 33776.465,E2 33776.465} C_VEL
LIN {X 0,Y 730.059,Z 827.946,A -85,B 0,C 180,E1 33775.384,E2 33775.384} C_VEL
LIN {X 0,Y 729.744,Z 849.07,A -85,B 0,C 180,E1 33774.185,E2 33774.185} C_VEL
LIN {X 0,Y 729.359,Z 868.79,A -85,B 0,C 180,E1 33772.889,E2 33772.889} C_VEL
LIN {X 0,Y 729.072,Z 887.765,A -85,B 0,C 180,E1 33771.48,E2 33771.48} C_VEL
LIN {X 0,Y 728.776,Z 904.462,A -85,B 0,C 180,E1 33770.06,E2 33770.06} C_VEL
LIN {X 0,Y 728.573,Z 920.962,A -85,B 0,C 180,E1 33768.483,E2 33768.483} C_VEL
LIN {X 0,Y 728.355,Z 935.453,A -85,B 0,C 180,E1 33766.893,E2 33766.893} C_VEL
LIN {X 0,Y 728.207,Z 949.058,A -85,B 0,C 180,E1 33765.204,E2 33765.204} C_VEL
LIN {X 0,Y 728.086,Z 960.794,A -85,B 0,C 180,E1 33763.501,E2 33763.501} C_VEL
LIN {X 0,Y 728.025,Z 970.951,A -85,B 0,C 180,E1 33761.808,E2 33761.808} C_VEL
LIN {X 0,Y 727.958,Z 980.182,A -85,B 0,C 180,E1 33759.966,E2 33759.966} C_VEL
LIN {X 0,Y 727.923,Z 986.815,A -85,B 0,C 180,E1 33758.372,E2 33758.372} C_VEL
LIN {X 0,Y 727.91,Z 993.245,A -85,B 0,C 180,E1 33756.467,E2 33756.467} C_VEL
LIN {X 0,Y 727.917,Z 997.813,A -85,B 0,C 180,E1 33754.57,E2 33754.57} C_VEL
LIN {X 0,Y 727.882,Z 1000.684,A -85,B 0,C 180,E1 33752.835,E2 33752.835} C_VEL
LIN {X 0,Y 727.89,Z 1002.262,A -85,B 0,C 180,E1 33750.866,E2 33750.866} C_VEL
LIN {X 0,Y 727.883,Z 1002.306,A -85,B 0,C 180,E1 33749.292,E2 33749.292} C_VEL
LIN {X 0,Y 727.89,Z 1001.017,A -85,B 0,C 180,E1 33747.402,E2 33747.402} C_VEL
LIN {X 0,Y 727.915,Z 997.971,A -85,B 0,C 180,E1 33745.509,E2 33745.509} C_VEL
LIN {X 0,Y 727.915,Z 993.864,A -85,B 0,C 180,E1 33743.77,E2 33743.77} C_VEL
LIN {X 0,Y 727.937,Z 987.422,A -85,B 0,C 180,E1 33741.787,E2 33741.787} C_VEL
LIN {X 0,Y 727.95,Z 980.891,A -85,B 0,C 180,E1 33740.193,E2 33740.193} C_VEL
LIN {X 0,Y 728.027,Z 971.868,A -85,B 0,C 180,E1 33738.352,E2 33738.352} C_VEL
LIN {X 0,Y 728.079,Z 961.315,A -85,B 0,C 180,E1 33736.58,E2 33736.58} C_VEL
LIN {X 0,Y 728.191,Z 950.217,A -85,B 0,C 180,E1 33734.958,E2 33734.958} C_VEL
LIN {X 0,Y 728.355,Z 936.633,A -85,B 0,C 180,E1 33733.244,E2 33733.244} C_VEL
LIN {X 0,Y 728.512,Z 923.292,A -85,B 0,C 180,E1 33731.764,E2 33731.764} C_VEL
LIN {X 0,Y 728.757,Z 906.319,A -85,B 0,C 180,E1 33730.107,E2 33730.107} C_VEL
LIN {X 0,Y 729.028,Z 889.791,A -85,B 0,C 180,E1 33728.687,E2 33728.687} C_VEL
LIN {X 0,Y 729.342,Z 870.252,A -85,B 0,C 180,E1 33727.214,E2 33727.214} C_VEL
LIN {X 0,Y 729.683,Z 851.761,A -85,B 0,C 180,E1 33725.985,E2 33725.985} C_VEL
LIN {X 0,Y 730.033,Z 830.348,A -85,B 0,C 180,E1 33724.745,E2 33724.745} C_VEL
LIN {X 0,Y 730.388,Z 810.156,A -85,B 0,C 180,E1 33723.726,E2 33723.726} C_VEL
LIN {X 0,Y 730.764,Z 786.714,A -85,B 0,C 180,E1 33722.718,E2 33722.718} C_VEL
LIN {X 0,Y 731.014,Z 766.425,A -85,B 0,C 180,E1 33721.976,E2 33721.976} C_VEL
LIN {X 0,Y 731.408,Z 740.95,A -85,B 0,C 180,E1 33721.214,E2 33721.214} C_VEL
LIN {X 0,Y 731.62,Z 719.758,A -85,B 0,C 180,E1 33720.713,E2 33720.713} C_VEL
LIN {X 0,Y 731.875,Z 695.743,A -85,B 0,C 180,E1 33720.277,E2 33720.277} C_VEL
LIN {X 0,Y 732.027,Z 654.274,A -85,B 0,C 180,E1 33719.79,E2 33719.79} C_VEL
LIN {X 0,Y 732.741,Z 411.97,A -85,B 0,C 180,E1 33717.092,E2 33717.092} C_VEL
LIN {X 0,Y 732.91,Z 302.894,A -85,B 0,C 180,E1 33715.845,E2 33715.845} C_VEL
LIN {X 0,Y 732.215,Z 298.171,A -85,B 0,C 180,E1 33715.739,E2 33715.739} C_VEL
LIN {X 0,Y 732.862,Z 239.016,A -85,B 0,C 180,E1 33713.063,E2 33713.063} C_VEL
LIN {X 0,Y 733.177,Z 205.822,A -85,B 0,C 180,E1 33711.519,E2 33711.519} C_VEL
LIN {X 0,Y 729.325,Z 197.843,A -85,B 0,C 180,E1 33710.894,E2 33710.894} C_VEL
LIN {X 0,Y 728.113,Z 194.537,A -85,B 0,C 180,E1 33710.638,E2 33710.638} C_VEL
LIN {X 0,Y 728.154,Z 194.53,A -85,B 0,C 180,E1 33707.744,E2 33707.744} C_VEL
LIN {X 0,Y 728.109,Z 194.535,A -85,B 0,C 180,E1 33704.767,E2 33704.767} C_VEL
LIN {X 0,Y 728.139,Z 194.532,A -85,B 0,C 180,E1 33702.02,E2 33702.02} C_VEL
LIN {X 0,Y 728.123,Z 194.534,A -85,B 0,C 180,E1 33699.074,E2 33699.074} C_VEL
LIN {X 0,Y 728.13,Z 194.534,A -85,B 0,C 180,E1 33696.285,E2 33696.285} C_VEL
LIN {X 0,Y 728.19,Z 194.734,A -85,B 0,C 180,E1 33693.478,E2 33693.478} C_VEL
LIN {X 0,Y 731.371,Z 203.57,A -85,B 0,C 180,E1 33692.776,E2 33692.776} C_VEL
LIN {X 0,Y 730.574,Z 253.886,A -85,B 0,C 180,E1 33689.93,E2 33689.93} C_VEL
LIN {X 0,Y 730.055,Z 312.143,A -85,B 0,C 180,E1 33686.749,E2 33686.749} C_VEL
LIN {X 0,Y 729.76,Z 365.856,A -85,B 0,C 180,E1 33683.884,E2 33683.884} C_VEL
LIN {X 0,Y 729.374,Z 419.681,A -85,B 0,C 180,E1 33681.05,E2 33681.05} C_VEL
LIN {X 0,Y 729.027,Z 470.287,A -85,B 0,C 180,E1 33678.424,E2 33678.424} C_VEL
LIN {X 0,Y 729.415,Z 478.267,A -85,B 0,C 180,E1 33678.333,E2 33678.333} C_VEL
LIN {X 0,Y 729.12,Z 679.864,A -85,B 0,C 180,E1 33676.281,E2 33676.281} C_VEL
LIN {X 0,Y 729.021,Z 698.948,A -85,B 0,C 180,E1 33675.937,E2 33675.937} C_VEL
LIN {X 0,Y 728.904,Z 717.095,A -85,B 0,C 180,E1 33675.464,E2 33675.464} C_VEL
LIN {X 0,Y 728.748,Z 734.427,A -85,B 0,C 180,E1 33674.867,E2 33674.867} C_VEL
LIN {X 0,Y 728.624,Z 751.176,A -85,B 0,C 180,E1 33674.139,E2 33674.139} C_VEL
LIN {X 0,Y 728.479,Z 766.812,A -85,B 0,C 180,E1 33673.306,E2 33673.306} C_VEL
LIN {X 0,Y 728.334,Z 781.987,A -85,B 0,C 180,E1 33672.326,E2 33672.326} C_VEL
LIN {X 0,Y 728.205,Z 795.921,A -85,B 0,C 180,E1 33671.244,E2 33671.244} C_VEL
LIN {X 0,Y 728.1,Z 808.747,A -85,B 0,C 180,E1 33670.044,E2 33670.044} C_VEL
LIN {X 0,Y 728.023,Z 820.005,A -85,B 0,C 180,E1 33668.769,E2 33668.769} C_VEL
LIN {X 0,Y 727.969,Z 829.898,A -85,B 0,C 180,E1 33667.39,E2 33667.39} C_VEL
LIN {X 0,Y 727.939,Z 837.852,A -85,B 0,C 180,E1 33665.992,E2 33665.992} C_VEL
LIN {X 0,Y 727.919,Z 844.042,A -85,B 0,C 180,E1 33664.57,E2 33664.57} C_VEL
LIN {X 0,Y 727.915,Z 848.464,A -85,B 0,C 180,E1 33663.15,E2 33663.15} C_VEL
LIN {X 0,Y 727.911,Z 851.339,A -85,B 0,C 180,E1 33661.653,E2 33661.653} C_VEL
LIN {X 0,Y 727.912,Z 852.449,A -85,B 0,C 180,E1 33660.157,E2 33660.157} C_VEL
LIN {X 0,Y 727.913,Z 851.82,A -85,B 0,C 180,E1 33658.662,E2 33658.662} C_VEL
LIN {X 0,Y 727.913,Z 849.437,A -85,B 0,C 180,E1 33657.165,E2 33657.165} C_VEL
LIN {X 0,Y 727.921,Z 845.235,A -85,B 0,C 180,E1 33655.667,E2 33655.667} C_VEL
LIN {X 0,Y 727.931,Z 839.464,A -85,B 0,C 180,E1 33654.245,E2 33654.245} C_VEL
LIN {X 0,Y 727.968,Z 831.804,A -85,B 0,C 180,E1 33652.82,E2 33652.82} C_VEL
LIN {X 0,Y 728.012,Z 822.466,A -85,B 0,C 180,E1 33651.451,E2 33651.451} C_VEL
LIN {X 0,Y 728.085,Z 811.922,A -85,B 0,C 180,E1 33650.195,E2 33650.195} C_VEL
LIN {X 0,Y 728.177,Z 799.737,A -85,B 0,C 180,E1 33648.997,E2 33648.997} C_VEL
LIN {X 0,Y 728.297,Z 785.992,A -85,B 0,C 180,E1 33647.874,E2 33647.874} C_VEL
LIN {X 0,Y 728.304,Z 784.724,A -85,B 0,C 180,E1 33647.782,E2 33647.782} C_VEL
LIN {X 0,Y 727.372,Z 779.122,A -85,B 0,C 180,E1 33647.367,E2 33647.367} C_VEL
LIN {X 0,Y 721.623,Z 764.762,A -85,B 0,C 180,E1 33646.353,E2 33646.353} C_VEL
LIN {X 0,Y 720.732,Z 758.498,A -85,B 0,C 180,E1 33645.987,E2 33645.987} C_VEL
LIN {X 0,Y 720.903,Z 741.804,A -85,B 0,C 180,E1 33645.181,E2 33645.181} C_VEL
LIN {X 0,Y 721.108,Z 724.487,A -85,B 0,C 180,E1 33644.513,E2 33644.513} C_VEL
LIN {X 0,Y 721.275,Z 705.803,A -85,B 0,C 180,E1 33643.96,E2 33643.96} C_VEL
LIN {X 0,Y 721.401,Z 686.903,A -85,B 0,C 180,E1 33643.561,E2 33643.561} C_VEL
LIN {X 0,Y 721.479,Z 666.781,A -85,B 0,C 180,E1 33643.296,E2 33643.296} C_VEL
LIN {X 0,Y 721.671,Z 473.025,A -85,B 0,C 180,E1 33641.319,E2 33641.319} C_VEL
LIN {X 0,Y 721.309,Z 469.724,A -85,B 0,C 180,E1 33641.261,E2 33641.261} C_VEL
LIN {X 0,Y 721.774,Z 418.133,A -85,B 0,C 180,E1 33638.548,E2 33638.548} C_VEL
LIN {X 0,Y 722.276,Z 363.537,A -85,B 0,C 180,E1 33635.632,E2 33635.632} C_VEL
LIN {X 0,Y 722.825,Z 311.685,A -85,B 0,C 180,E1 33632.807,E2 33632.807} C_VEL
LIN {X 0,Y 723.408,Z 258.979,A -85,B 0,C 180,E1 33629.885,E2 33629.885} C_VEL
LIN {X 0,Y 724.003,Z 208.72,A -85,B 0,C 180,E1 33627.034,E2 33627.034} C_VEL
LIN {X 0,Y 723.758,Z 205.468,A -85,B 0,C 180,E1 33626.833,E2 33626.833} C_VEL
LIN {X 0,Y 720.196,Z 195.523,A -85,B 0,C 180,E1 33626.05,E2 33626.05} C_VEL
LIN {X 0,Y 720.182,Z 195.518,A -85,B 0,C 180,E1 33623.245,E2 33623.245} C_VEL
LIN {X 0,Y 720.214,Z 195.521,A -85,B 0,C 180,E1 33620.401,E2 33620.401} C_VEL
